  PROC DrawPart118()
    MoveL Offs(pOrigin,175.68,196.88,0.00),v40,fine,tPen\WObj:=wPaper;
    MoveL Offs(pOrigin,175.68,196.88,6.00),v60,z5,tPen\WObj:=wPaper;
    MoveL Offs(pOrigin,176.60,194.01,6.00),vTravel,z5,tPen\WObj:=wPaper;
    MoveL Offs(pOrigin,176.60,194.01,0.00),v60,z0,tPen\WObj:=wPaper;
    MoveL Offs(pOrigin,168.94,201.68,0.00),v40,z0,tPen\WObj:=wPaper;
    MoveL Offs(pOrigin,169.41,202.55,0.00),v40,z0,tPen\WObj:=wPaper;
    MoveL Offs(pOrigin,171.06,204.21,0.00),v40,fine,tPen\WObj:=wPaper;
    MoveL Offs(pOrigin,171.06,204.21,6.00),v60,z5,tPen\WObj:=wPaper;
    MoveL Offs(pOrigin,168.81,204.95,6.00),vTravel,z5,tPen\WObj:=wPaper;
    MoveL Offs(pOrigin,168.81,204.95,0.00),v60,z0,tPen\WObj:=wPaper;
    MoveL Offs(pOrigin,170.47,206.60,0.00),v40,z0,tPen\WObj:=wPaper;
    MoveL Offs(pOrigin,170.87,207.21,0.00),v40,z0,tPen\WObj:=wPaper;
    MoveL Offs(pOrigin,163.66,214.42,0.00),v40,z0,tPen\WObj:=wPaper;
    MoveL Offs(pOrigin,164.35,213.92,0.00),v40,z0,tPen\WObj:=wPaper;
    MoveL Offs(pOrigin,166.30,215.88,0.00),v40,fine,tPen\WObj:=wPaper;
    MoveL Offs(pOrigin,166.30,215.88,6.00),v60,z5,tPen\WObj:=wPaper;
    MoveL Offs(pOrigin,167.65,215.73,6.00),vTravel,z5,tPen\WObj:=wPaper;
    MoveL Offs(pOrigin,167.65,215.73,0.00),v60,z0,tPen\WObj:=wPaper;
    MoveL Offs(pOrigin,170.05,218.13,0.00),v40,z0,tPen\WObj:=wPaper;
    MoveL Offs(pOrigin,170.39,218.15,0.00),v40,z0,tPen\WObj:=wPaper;
    MoveL Offs(pOrigin,163.02,225.51,0.00),v40,z0,tPen\WObj:=wPaper;
    MoveL Offs(pOrigin,163.94,225.14,0.00),v40,z0,tPen\WObj:=wPaper;
    MoveL Offs(pOrigin,165.21,225.14,0.00),v40,z0,tPen\WObj:=wPaper;
    MoveL Offs(pOrigin,165.00,224.51,0.00),v40,z0,tPen\WObj:=wPaper;
    MoveL Offs(pOrigin,165.21,224.94,0.00),v40,z0,tPen\WObj:=wPaper;
    MoveL Offs(pOrigin,165.00,224.51,0.00),v40,z0,tPen\WObj:=wPaper;
    MoveL Offs(pOrigin,164.58,224.09,0.00),v40,z0,tPen\WObj:=wPaper;
    MoveL Offs(pOrigin,163.51,224.09,0.00),v40,z0,tPen\WObj:=wPaper;
    MoveL Offs(pOrigin,163.09,224.51,0.00),v40,z0,tPen\WObj:=wPaper;
    MoveL Offs(pOrigin,163.30,224.94,0.00),v40,z0,tPen\WObj:=wPaper;
    MoveL Offs(pOrigin,163.09,224.51,0.00),v40,z0,tPen\WObj:=wPaper;
    MoveL Offs(pOrigin,162.73,224.25,0.00),v40,z0,tPen\WObj:=wPaper;
    MoveL Offs(pOrigin,170.99,232.52,0.00),v40,z0,tPen\WObj:=wPaper;
    MoveL Offs(pOrigin,170.74,232.16,0.00),v40,z0,tPen\WObj:=wPaper;
    MoveL Offs(pOrigin,171.16,232.38,0.00),v40,z0,tPen\WObj:=wPaper;
    MoveL Offs(pOrigin,170.74,232.16,0.00),v40,z0,tPen\WObj:=wPaper;
    MoveL Offs(pOrigin,170.64,232.83,0.00),v40,z0,tPen\WObj:=wPaper;
    MoveL Offs(pOrigin,175.15,228.32,0.00),v40,z0,tPen\WObj:=wPaper;
    MoveL Offs(pOrigin,175.20,228.98,0.00),v40,z0,tPen\WObj:=wPaper;
    MoveL Offs(pOrigin,175.84,229.61,0.00),v40,z0,tPen\WObj:=wPaper;
    MoveL Offs(pOrigin,175.20,228.98,0.00),v40,z0,tPen\WObj:=wPaper;
    MoveL Offs(pOrigin,175.20,229.37,0.00),v40,z0,tPen\WObj:=wPaper;
    MoveL Offs(pOrigin,173.71,229.37,0.00),v40,z0,tPen\WObj:=wPaper;
    MoveL Offs(pOrigin,173.71,230.04,0.00),v40,z0,tPen\WObj:=wPaper;
    MoveL Offs(pOrigin,174.14,230.25,0.00),v40,z0,tPen\WObj:=wPaper;
    MoveL Offs(pOrigin,173.71,230.04,0.00),v40,z0,tPen\WObj:=wPaper;
    MoveL Offs(pOrigin,174.35,230.46,0.00),v40,z0,tPen\WObj:=wPaper;
    MoveL Offs(pOrigin,174.77,230.89,0.00),v40,z0,tPen\WObj:=wPaper;
    MoveL Offs(pOrigin,174.35,230.46,0.00),v40,z0,tPen\WObj:=wPaper;
    MoveL Offs(pOrigin,174.78,230.42,0.00),v40,z0,tPen\WObj:=wPaper;
    MoveL Offs(pOrigin,176.69,230.42,0.00),v40,z0,tPen\WObj:=wPaper;
    MoveL Offs(pOrigin,176.94,229.51,0.00),v40,z0,tPen\WObj:=wPaper;
    MoveL Offs(pOrigin,172.74,233.72,0.00),v40,z0,tPen\WObj:=wPaper;
    MoveL Offs(pOrigin,173.71,233.65,0.00),v40,z0,tPen\WObj:=wPaper;
    MoveL Offs(pOrigin,174.14,233.86,0.00),v40,z0,tPen\WObj:=wPaper;
    MoveL Offs(pOrigin,173.71,233.65,0.00),v40,z0,tPen\WObj:=wPaper;
    MoveL Offs(pOrigin,173.63,234.32,0.00),v40,z0,tPen\WObj:=wPaper;
    MoveL Offs(pOrigin,177.84,230.11,0.00),v40,z0,tPen\WObj:=wPaper;
    MoveL Offs(pOrigin,178.74,230.71,0.00),v40,z0,tPen\WObj:=wPaper;
    MoveL Offs(pOrigin,174.68,234.76,0.00),v40,z0,tPen\WObj:=wPaper;
    MoveL Offs(pOrigin,174.15,234.18,0.00),v40,z0,tPen\WObj:=wPaper;
    MoveL Offs(pOrigin,161.22,221.25,0.00),v40,z0,tPen\WObj:=wPaper;
    MoveL Offs(pOrigin,161.09,221.47,0.00),v40,z0,tPen\WObj:=wPaper;
    MoveL Offs(pOrigin,170.25,212.31,0.00),v40,z0,tPen\WObj:=wPaper;
    MoveL Offs(pOrigin,169.88,211.99,0.00),v40,z0,tPen\WObj:=wPaper;
    MoveL Offs(pOrigin,168.08,210.19,0.00),v40,fine,tPen\WObj:=wPaper;
    MoveL Offs(pOrigin,168.08,210.19,6.00),v60,z5,tPen\WObj:=wPaper;
    MoveL Offs(pOrigin,167.93,211.54,6.00),vTravel,z5,tPen\WObj:=wPaper;
    MoveL Offs(pOrigin,167.93,211.54,0.00),v60,z0,tPen\WObj:=wPaper;
    MoveL Offs(pOrigin,169.89,213.49,0.00),v40,z0,tPen\WObj:=wPaper;
    MoveL Offs(pOrigin,170.25,213.81,0.00),v40,z0,tPen\WObj:=wPaper;
    MoveL Offs(pOrigin,161.38,222.67,0.00),v40,fine,tPen\WObj:=wPaper;
    MoveL Offs(pOrigin,161.38,222.67,6.00),v60,z5,tPen\WObj:=wPaper;
    MoveL Offs(pOrigin,162.45,221.98,6.00),vTravel,z5,tPen\WObj:=wPaper;
    MoveL Offs(pOrigin,162.45,221.98,0.00),v60,z0,tPen\WObj:=wPaper;
    MoveL Offs(pOrigin,163.51,221.98,0.00),v40,z0,tPen\WObj:=wPaper;
    MoveL Offs(pOrigin,163.09,220.92,0.00),v40,z0,tPen\WObj:=wPaper;
    MoveL Offs(pOrigin,162.02,220.92,0.00),v40,fine,tPen\WObj:=wPaper;
    MoveL Offs(pOrigin,162.02,220.92,6.00),v60,z5,tPen\WObj:=wPaper;
    MoveL Offs(pOrigin,165.27,220.82,6.00),vTravel,z5,tPen\WObj:=wPaper;
    MoveL Offs(pOrigin,165.27,220.82,0.00),v60,z0,tPen\WObj:=wPaper;
    MoveL Offs(pOrigin,168.12,223.67,0.00),v40,fine,tPen\WObj:=wPaper;
    MoveL Offs(pOrigin,168.12,223.67,6.00),v60,z5,tPen\WObj:=wPaper;
    MoveL Offs(pOrigin,166.70,223.45,6.00),vTravel,z5,tPen\WObj:=wPaper;
    MoveL Offs(pOrigin,166.70,223.45,0.00),v60,z0,tPen\WObj:=wPaper;
    MoveL Offs(pOrigin,166.91,223.88,0.00),v40,z0,tPen\WObj:=wPaper;
    MoveL Offs(pOrigin,166.70,223.45,0.00),v40,z0,tPen\WObj:=wPaper;
    MoveL Offs(pOrigin,165.87,222.91,0.00),v40,z0,tPen\WObj:=wPaper;
    MoveL Offs(pOrigin,168.73,225.77,0.00),v40,z0,tPen\WObj:=wPaper;
    MoveL Offs(pOrigin,168.40,225.79,0.00),v40,z0,tPen\WObj:=wPaper;
    MoveL Offs(pOrigin,168.40,224.94,0.00),v40,z0,tPen\WObj:=wPaper;
    MoveL Offs(pOrigin,166.91,221.11,0.00),v40,z0,tPen\WObj:=wPaper;
    MoveL Offs(pOrigin,166.06,216.86,0.00),v40,z0,tPen\WObj:=wPaper;
    MoveL Offs(pOrigin,165.85,209.64,0.00),v40,z0,tPen\WObj:=wPaper;
    MoveL Offs(pOrigin,166.70,202.20,0.00),v40,z0,tPen\WObj:=wPaper;
    MoveL Offs(pOrigin,168.26,196.32,0.00),v40,z0,tPen\WObj:=wPaper;
    MoveL Offs(pOrigin,168.61,196.25,0.00),v40,z0,tPen\WObj:=wPaper;
    MoveL Offs(pOrigin,171.16,197.31,0.00),v40,z0,tPen\WObj:=wPaper;
    MoveL Offs(pOrigin,169.04,205.18,0.00),v40,z0,tPen\WObj:=wPaper;
    MoveL Offs(pOrigin,167.98,212.82,0.00),v40,z0,tPen\WObj:=wPaper;
    MoveL Offs(pOrigin,168.19,217.93,0.00),v40,z0,tPen\WObj:=wPaper;
    MoveL Offs(pOrigin,169.60,223.88,0.00),v40,z0,tPen\WObj:=wPaper;
    MoveL Offs(pOrigin,171.80,227.70,0.00),v40,z0,tPen\WObj:=wPaper;
    MoveL Offs(pOrigin,174.77,230.68,0.00),v40,z0,tPen\WObj:=wPaper;
    MoveL Offs(pOrigin,178.81,232.87,0.00),v40,z0,tPen\WObj:=wPaper;
    MoveL Offs(pOrigin,182.85,234.07,0.00),v40,z0,tPen\WObj:=wPaper;
    MoveL Offs(pOrigin,183.70,233.86,0.00),v40,z0,tPen\WObj:=wPaper;
    MoveL Offs(pOrigin,183.70,233.86,0.00),v40,z0,tPen\WObj:=wPaper;
    MoveL Offs(pOrigin,186.68,234.50,0.00),v40,z0,tPen\WObj:=wPaper;
    MoveL Offs(pOrigin,186.66,234.73,0.00),v40,z0,tPen\WObj:=wPaper;
    MoveL Offs(pOrigin,183.81,237.58,0.00),v40,z0,tPen\WObj:=wPaper;
    MoveL Offs(pOrigin,184.34,236.76,0.00),v40,z0,tPen\WObj:=wPaper;
    MoveL Offs(pOrigin,189.86,236.76,0.00),v40,z0,tPen\WObj:=wPaper;
    MoveL Offs(pOrigin,189.88,236.47,0.00),v40,z0,tPen\WObj:=wPaper;
    MoveL Offs(pOrigin,192.44,239.02,0.00),v40,z0,tPen\WObj:=wPaper;
    MoveL Offs(pOrigin,192.49,239.35,0.00),v40,z0,tPen\WObj:=wPaper;
    MoveL Offs(pOrigin,195.05,236.80,0.00),v40,z0,tPen\WObj:=wPaper;
    MoveL Offs(pOrigin,195.43,237.54,0.00),v40,z0,tPen\WObj:=wPaper;
    MoveL Offs(pOrigin,197.98,240.09,0.00),v40,z0,tPen\WObj:=wPaper;
    MoveL Offs(pOrigin,197.43,240.39,0.00),v40,z0,tPen\WObj:=wPaper;
  ENDPROC

  PROC DrawPart119()
    MoveL Offs(pOrigin,204.49,233.32,0.00),v40,z0,tPen\WObj:=wPaper;
    MoveL Offs(pOrigin,204.10,232.77,0.00),v40,z0,tPen\WObj:=wPaper;
    MoveL Offs(pOrigin,202.30,230.97,0.00),v40,z0,tPen\WObj:=wPaper;
    MoveL Offs(pOrigin,203.04,230.42,0.00),v40,z0,tPen\WObj:=wPaper;
    MoveL Offs(pOrigin,204.10,230.42,0.00),v40,z0,tPen\WObj:=wPaper;
    MoveL Offs(pOrigin,204.69,230.37,0.00),v40,z0,tPen\WObj:=wPaper;
    MoveL Offs(pOrigin,203.34,229.02,0.00),v40,z0,tPen\WObj:=wPaper;
    MoveL Offs(pOrigin,203.46,229.37,0.00),v40,z0,tPen\WObj:=wPaper;
    MoveL Offs(pOrigin,204.74,229.37,0.00),v40,z0,tPen\WObj:=wPaper;
    MoveL Offs(pOrigin,205.38,228.76,0.00),v40,z0,tPen\WObj:=wPaper;
    MoveL Offs(pOrigin,204.74,229.40,0.00),v40,z0,tPen\WObj:=wPaper;
    MoveL Offs(pOrigin,205.38,228.76,0.00),v40,fine,tPen\WObj:=wPaper;
    MoveL Offs(pOrigin,205.38,228.76,6.00),v60,z5,tPen\WObj:=wPaper;
    MoveL Offs(pOrigin,204.31,227.91,6.00),vTravel,z5,tPen\WObj:=wPaper;
    MoveL Offs(pOrigin,204.31,227.91,0.00),v60,z0,tPen\WObj:=wPaper;
    MoveL Offs(pOrigin,203.89,228.34,0.00),v40,z0,tPen\WObj:=wPaper;
    MoveL Offs(pOrigin,204.31,227.91,0.00),v40,z0,tPen\WObj:=wPaper;
    MoveL Offs(pOrigin,204.68,227.38,0.00),v40,z0,tPen\WObj:=wPaper;
    MoveL Offs(pOrigin,208.44,231.13,0.00),v40,z0,tPen\WObj:=wPaper;
    MoveL Offs(pOrigin,208.69,232.11,0.00),v40,z0,tPen\WObj:=wPaper;
    MoveL Offs(pOrigin,205.99,234.82,0.00),v40,fine,tPen\WObj:=wPaper;
    MoveL Offs(pOrigin,205.99,234.82,6.00),v60,z5,tPen\WObj:=wPaper;
    MoveL Offs(pOrigin,205.98,236.32,6.00),vTravel,z5,tPen\WObj:=wPaper;
    MoveL Offs(pOrigin,205.98,236.32,0.00),v60,z0,tPen\WObj:=wPaper;
    MoveL Offs(pOrigin,208.24,234.06,0.00),v40,z0,tPen\WObj:=wPaper;
    MoveL Offs(pOrigin,207.85,233.53,0.00),v40,z0,tPen\WObj:=wPaper;
    MoveL Offs(pOrigin,206.95,232.63,0.00),v40,z0,tPen\WObj:=wPaper;
    MoveL Offs(pOrigin,207.29,232.38,0.00),v40,z0,tPen\WObj:=wPaper;
    MoveL Offs(pOrigin,207.71,228.76,0.00),v40,z0,tPen\WObj:=wPaper;
    MoveL Offs(pOrigin,207.29,228.34,0.00),v40,z0,tPen\WObj:=wPaper;
    MoveL Offs(pOrigin,206.44,228.34,0.00),v40,z0,tPen\WObj:=wPaper;
    MoveL Offs(pOrigin,204.95,229.40,0.00),v40,z0,tPen\WObj:=wPaper;
    MoveL Offs(pOrigin,204.03,231.10,0.00),v40,z0,tPen\WObj:=wPaper;
    MoveL Offs(pOrigin,203.68,232.38,0.00),v40,z0,tPen\WObj:=wPaper;
    MoveL Offs(pOrigin,203.46,236.41,0.00),v40,z0,tPen\WObj:=wPaper;
    MoveL Offs(pOrigin,202.47,240.66,0.00),v40,z0,tPen\WObj:=wPaper;
    MoveL Offs(pOrigin,200.98,244.91,0.00),v40,z0,tPen\WObj:=wPaper;
    MoveL Offs(pOrigin,196.80,252.14,0.00),v40,z0,tPen\WObj:=wPaper;
    MoveL Offs(pOrigin,196.24,254.48,0.00),v40,z0,tPen\WObj:=wPaper;
    MoveL Offs(pOrigin,196.24,258.30,0.00),v40,z0,tPen\WObj:=wPaper;
    MoveL Offs(pOrigin,196.80,260.42,0.00),v40,z0,tPen\WObj:=wPaper;
    MoveL Offs(pOrigin,197.73,262.12,0.00),v40,z0,tPen\WObj:=wPaper;
    MoveL Offs(pOrigin,199.00,263.12,0.00),v40,z0,tPen\WObj:=wPaper;
    MoveL Offs(pOrigin,200.70,263.19,0.00),v40,z0,tPen\WObj:=wPaper;
    MoveL Offs(pOrigin,201.98,261.91,0.00),v40,z0,tPen\WObj:=wPaper;
    MoveL Offs(pOrigin,201.98,261.91,0.00),v40,z0,tPen\WObj:=wPaper;
    MoveL Offs(pOrigin,202.54,261.70,0.00),v40,z0,tPen\WObj:=wPaper;
    MoveL Offs(pOrigin,202.90,260.00,0.00),v40,z0,tPen\WObj:=wPaper;
    MoveL Offs(pOrigin,203.46,259.36,0.00),v40,z0,tPen\WObj:=wPaper;
    MoveL Offs(pOrigin,203.68,258.09,0.00),v40,z0,tPen\WObj:=wPaper;
    MoveL Offs(pOrigin,203.39,257.02,0.00),v40,z0,tPen\WObj:=wPaper;
    MoveL Offs(pOrigin,204.38,252.14,0.00),v40,z0,tPen\WObj:=wPaper;
    MoveL Offs(pOrigin,205.02,250.44,0.00),v40,z0,tPen\WObj:=wPaper;
    MoveL Offs(pOrigin,205.80,250.65,0.00),v40,z0,tPen\WObj:=wPaper;
    MoveL Offs(pOrigin,205.93,250.44,0.00),v40,z0,tPen\WObj:=wPaper;
    MoveL Offs(pOrigin,205.93,260.42,0.00),v40,z0,tPen\WObj:=wPaper;
    MoveL Offs(pOrigin,206.23,260.85,0.00),v40,z0,tPen\WObj:=wPaper;
    MoveL Offs(pOrigin,206.01,261.27,0.00),v40,z0,tPen\WObj:=wPaper;
    MoveL Offs(pOrigin,206.23,260.85,0.00),v40,z0,tPen\WObj:=wPaper;
    MoveL Offs(pOrigin,206.01,261.05,0.00),v40,z0,tPen\WObj:=wPaper;
    MoveL Offs(pOrigin,203.04,261.05,0.00),v40,z0,tPen\WObj:=wPaper;
    MoveL Offs(pOrigin,203.04,259.99,0.00),v40,z0,tPen\WObj:=wPaper;
    MoveL Offs(pOrigin,207.29,259.99,0.00),v40,z0,tPen\WObj:=wPaper;
    MoveL Offs(pOrigin,207.78,260.34,0.00),v40,z0,tPen\WObj:=wPaper;
    MoveL Offs(pOrigin,203.12,255.69,0.00),v40,z0,tPen\WObj:=wPaper;
    MoveL Offs(pOrigin,203.68,255.77,0.00),v40,z0,tPen\WObj:=wPaper;
    MoveL Offs(pOrigin,207.08,255.77,0.00),v40,z0,tPen\WObj:=wPaper;
    MoveL Offs(pOrigin,207.08,254.71,0.00),v40,z0,tPen\WObj:=wPaper;
    MoveL Offs(pOrigin,203.89,254.71,0.00),v40,z0,tPen\WObj:=wPaper;
    MoveL Offs(pOrigin,203.42,254.49,0.00),v40,z0,tPen\WObj:=wPaper;
    MoveL Offs(pOrigin,208.23,259.30,0.00),v40,z0,tPen\WObj:=wPaper;
    MoveL Offs(pOrigin,207.93,258.94,0.00),v40,z0,tPen\WObj:=wPaper;
    MoveL Offs(pOrigin,207.07,258.73,0.00),v40,z0,tPen\WObj:=wPaper;
    MoveL Offs(pOrigin,207.29,257.88,0.00),v40,z0,tPen\WObj:=wPaper;
    MoveL Offs(pOrigin,207.07,257.88,0.00),v40,z0,tPen\WObj:=wPaper;
    MoveL Offs(pOrigin,207.50,257.88,0.00),v40,z0,tPen\WObj:=wPaper;
    MoveL Offs(pOrigin,203.04,257.88,0.00),v40,z0,tPen\WObj:=wPaper;
    MoveL Offs(pOrigin,203.25,257.45,0.00),v40,z0,tPen\WObj:=wPaper;
    MoveL Offs(pOrigin,202.12,258.51,0.00),v40,z0,tPen\WObj:=wPaper;
    MoveL Offs(pOrigin,201.98,259.79,0.00),v40,z0,tPen\WObj:=wPaper;
    MoveL Offs(pOrigin,202.61,258.94,0.00),v40,z0,tPen\WObj:=wPaper;
    MoveL Offs(pOrigin,207.50,258.94,0.00),v40,fine,tPen\WObj:=wPaper;
    MoveL Offs(pOrigin,207.50,258.94,6.00),v60,z5,tPen\WObj:=wPaper;
    MoveL Offs(pOrigin,208.76,258.93,6.00),vTravel,z5,tPen\WObj:=wPaper;
    MoveL Offs(pOrigin,208.76,258.93,0.00),v60,z0,tPen\WObj:=wPaper;
    MoveL Offs(pOrigin,194.18,273.50,0.00),v40,z0,tPen\WObj:=wPaper;
    MoveL Offs(pOrigin,194.64,274.08,0.00),v40,z0,tPen\WObj:=wPaper;
    MoveL Offs(pOrigin,204.71,284.15,0.00),v40,z0,tPen\WObj:=wPaper;
    MoveL Offs(pOrigin,204.31,284.28,0.00),v40,z0,tPen\WObj:=wPaper;
    MoveL Offs(pOrigin,191.35,284.28,0.00),v40,z0,tPen\WObj:=wPaper;
    MoveL Offs(pOrigin,190.93,283.81,0.00),v40,z0,tPen\WObj:=wPaper;
    MoveL Offs(pOrigin,195.58,288.47,0.00),v40,fine,tPen\WObj:=wPaper;
    MoveL Offs(pOrigin,195.58,288.47,6.00),v60,z5,tPen\WObj:=wPaper;
    MoveL Offs(pOrigin,193.90,289.54,6.00),vTravel,z5,tPen\WObj:=wPaper;
    MoveL Offs(pOrigin,193.90,289.54,0.00),v60,z0,tPen\WObj:=wPaper;
    MoveL Offs(pOrigin,194.11,289.96,0.00),v40,z0,tPen\WObj:=wPaper;
    MoveL Offs(pOrigin,193.90,289.54,0.00),v40,z0,tPen\WObj:=wPaper;
    MoveL Offs(pOrigin,193.48,289.56,0.00),v40,z0,tPen\WObj:=wPaper;
    MoveL Offs(pOrigin,191.56,289.56,0.00),v40,z0,tPen\WObj:=wPaper;
    MoveL Offs(pOrigin,191.09,289.95,0.00),v40,z0,tPen\WObj:=wPaper;
    MoveL Offs(pOrigin,196.20,295.06,0.00),v40,z0,tPen\WObj:=wPaper;
    MoveL Offs(pOrigin,196.45,295.49,0.00),v40,z0,tPen\WObj:=wPaper;
    MoveL Offs(pOrigin,197.51,297.19,0.00),v40,z0,tPen\WObj:=wPaper;
    MoveL Offs(pOrigin,199.64,299.31,0.00),v40,z0,tPen\WObj:=wPaper;
    MoveL Offs(pOrigin,200.71,299.57,0.00),v40,z0,tPen\WObj:=wPaper;
    MoveL Offs(pOrigin,225.80,324.66,0.00),v40,fine,tPen\WObj:=wPaper;
    MoveL Offs(pOrigin,225.80,324.66,6.00),v60,z5,tPen\WObj:=wPaper;
    MoveL Offs(pOrigin,225.95,323.31,6.00),vTravel,z5,tPen\WObj:=wPaper;
    MoveL Offs(pOrigin,225.95,323.31,0.00),v60,z0,tPen\WObj:=wPaper;
    MoveL Offs(pOrigin,201.76,299.12,0.00),v40,z0,tPen\WObj:=wPaper;
    MoveL Offs(pOrigin,202.40,299.95,0.00),v40,z0,tPen\WObj:=wPaper;
    MoveL Offs(pOrigin,204.95,301.01,0.00),v40,z0,tPen\WObj:=wPaper;
    MoveL Offs(pOrigin,204.88,300.80,0.00),v40,z0,tPen\WObj:=wPaper;
    MoveL Offs(pOrigin,204.88,301.86,0.00),v40,fine,tPen\WObj:=wPaper;
    MoveL Offs(pOrigin,204.88,301.86,6.00),v60,z5,tPen\WObj:=wPaper;
    MoveL Offs(pOrigin,203.68,302.23,6.00),vTravel,z5,tPen\WObj:=wPaper;
    MoveL Offs(pOrigin,203.68,302.23,0.00),v60,z0,tPen\WObj:=wPaper;
    MoveL Offs(pOrigin,210.48,302.23,0.00),v40,fine,tPen\WObj:=wPaper;
    MoveL Offs(pOrigin,210.48,302.23,6.00),v60,z5,tPen\WObj:=wPaper;
    MoveL Offs(pOrigin,211.33,301.16,6.00),vTravel,z5,tPen\WObj:=wPaper;
  ENDPROC

  PROC DrawPart120()
    MoveL Offs(pOrigin,211.33,301.16,0.00),v60,z0,tPen\WObj:=wPaper;
    MoveL Offs(pOrigin,195.70,316.79,0.00),v40,z0,tPen\WObj:=wPaper;
    MoveL Offs(pOrigin,196.45,317.59,0.00),v40,z0,tPen\WObj:=wPaper;
    MoveL Offs(pOrigin,196.66,318.01,0.00),v40,z0,tPen\WObj:=wPaper;
    MoveL Offs(pOrigin,196.45,317.59,0.00),v40,z0,tPen\WObj:=wPaper;
    MoveL Offs(pOrigin,196.15,317.84,0.00),v40,z0,tPen\WObj:=wPaper;
    MoveL Offs(pOrigin,212.07,301.91,0.00),v40,z0,tPen\WObj:=wPaper;
    MoveL Offs(pOrigin,212.82,302.66,0.00),v40,z0,tPen\WObj:=wPaper;
    MoveL Offs(pOrigin,202.60,312.87,0.00),v40,z0,tPen\WObj:=wPaper;
    MoveL Offs(pOrigin,203.05,313.92,0.00),v40,z0,tPen\WObj:=wPaper;
    MoveL Offs(pOrigin,197.34,319.63,0.00),v40,z0,tPen\WObj:=wPaper;
    MoveL Offs(pOrigin,197.73,319.50,0.00),v40,z0,tPen\WObj:=wPaper;
    MoveL Offs(pOrigin,198.15,319.92,0.00),v40,z0,tPen\WObj:=wPaper;
    MoveL Offs(pOrigin,197.73,319.50,0.00),v40,z0,tPen\WObj:=wPaper;
    MoveL Offs(pOrigin,198.15,319.13,0.00),v40,z0,tPen\WObj:=wPaper;
    MoveL Offs(pOrigin,199.42,319.13,0.00),v40,z0,tPen\WObj:=wPaper;
    MoveL Offs(pOrigin,199.43,319.08,0.00),v40,z0,tPen\WObj:=wPaper;
    MoveL Offs(pOrigin,200.06,319.71,0.00),v40,z0,tPen\WObj:=wPaper;
    MoveL Offs(pOrigin,199.43,319.08,0.00),v40,z0,tPen\WObj:=wPaper;
    MoveL Offs(pOrigin,199.00,320.18,0.00),v40,z0,tPen\WObj:=wPaper;
    MoveL Offs(pOrigin,200.91,320.18,0.00),v40,z0,tPen\WObj:=wPaper;
    MoveL Offs(pOrigin,200.70,320.14,0.00),v40,z0,tPen\WObj:=wPaper;
    MoveL Offs(pOrigin,201.12,320.35,0.00),v40,z0,tPen\WObj:=wPaper;
    MoveL Offs(pOrigin,200.70,320.14,0.00),v40,fine,tPen\WObj:=wPaper;
    MoveL Offs(pOrigin,200.70,320.14,6.00),v60,z5,tPen\WObj:=wPaper;
    MoveL Offs(pOrigin,199.85,321.24,6.00),vTravel,z5,tPen\WObj:=wPaper;
    MoveL Offs(pOrigin,199.85,321.24,0.00),v60,z0,tPen\WObj:=wPaper;
    MoveL Offs(pOrigin,202.40,321.24,0.00),v40,z0,tPen\WObj:=wPaper;
    MoveL Offs(pOrigin,202.61,321.41,0.00),v40,z0,tPen\WObj:=wPaper;
    MoveL Offs(pOrigin,204.10,321.13,0.00),v40,z0,tPen\WObj:=wPaper;
    MoveL Offs(pOrigin,205.38,321.62,0.00),v40,z0,tPen\WObj:=wPaper;
    MoveL Offs(pOrigin,205.45,321.41,0.00),v40,z0,tPen\WObj:=wPaper;
    MoveL Offs(pOrigin,206.65,320.56,0.00),v40,z0,tPen\WObj:=wPaper;
    MoveL Offs(pOrigin,209.34,320.35,0.00),v40,z0,tPen\WObj:=wPaper;
    MoveL Offs(pOrigin,208.56,321.41,0.00),v40,z0,tPen\WObj:=wPaper;
    MoveL Offs(pOrigin,206.23,321.84,0.00),v40,z0,tPen\WObj:=wPaper;
    MoveL Offs(pOrigin,205.45,321.41,0.00),v40,z0,tPen\WObj:=wPaper;
    MoveL Offs(pOrigin,205.38,320.99,0.00),v40,z0,tPen\WObj:=wPaper;
    MoveL Offs(pOrigin,204.10,320.85,0.00),v40,z0,tPen\WObj:=wPaper;
    MoveL Offs(pOrigin,203.46,320.21,0.00),v40,z0,tPen\WObj:=wPaper;
    MoveL Offs(pOrigin,200.63,318.65,0.00),v40,z0,tPen\WObj:=wPaper;
    MoveL Offs(pOrigin,200.49,317.80,0.00),v40,z0,tPen\WObj:=wPaper;
    MoveL Offs(pOrigin,200.49,317.80,0.00),v40,z0,tPen\WObj:=wPaper;
    MoveL Offs(pOrigin,201.76,318.01,0.00),v40,z0,tPen\WObj:=wPaper;
    MoveL Offs(pOrigin,201.76,318.01,0.00),v40,z0,tPen\WObj:=wPaper;
    MoveL Offs(pOrigin,202.40,319.08,0.00),v40,z0,tPen\WObj:=wPaper;
    MoveL Offs(pOrigin,202.40,319.50,0.00),v40,z0,tPen\WObj:=wPaper;
    MoveL Offs(pOrigin,203.04,319.08,0.00),v40,z0,tPen\WObj:=wPaper;
    MoveL Offs(pOrigin,206.01,320.00,0.00),v40,z0,tPen\WObj:=wPaper;
    MoveL Offs(pOrigin,206.44,320.56,0.00),v40,z0,tPen\WObj:=wPaper;
    MoveL Offs(pOrigin,206.33,319.60,0.00),v40,z0,tPen\WObj:=wPaper;
    MoveL Offs(pOrigin,201.67,324.26,0.00),v40,z0,tPen\WObj:=wPaper;
    MoveL Offs(pOrigin,200.92,323.51,0.00),v40,z0,tPen\WObj:=wPaper;
    MoveL Offs(pOrigin,217.60,306.84,0.00),v40,z0,tPen\WObj:=wPaper;
    MoveL Offs(pOrigin,217.66,307.56,0.00),v40,z0,tPen\WObj:=wPaper;
    MoveL Offs(pOrigin,234.19,324.09,0.00),v40,z0,tPen\WObj:=wPaper;
    MoveL Offs(pOrigin,234.70,323.35,0.00),v40,z0,tPen\WObj:=wPaper;
    MoveL Offs(pOrigin,239.16,323.35,0.00),v40,z0,tPen\WObj:=wPaper;
    MoveL Offs(pOrigin,239.59,323.11,0.00),v40,z0,tPen\WObj:=wPaper;
    MoveL Offs(pOrigin,237.04,320.77,0.00),v40,z0,tPen\WObj:=wPaper;
    MoveL Offs(pOrigin,237.04,320.77,0.00),v40,z0,tPen\WObj:=wPaper;
    MoveL Offs(pOrigin,235.76,321.41,0.00),v40,z0,tPen\WObj:=wPaper;
    MoveL Offs(pOrigin,235.55,322.05,0.00),v40,z0,tPen\WObj:=wPaper;
    MoveL Offs(pOrigin,235.55,322.05,0.00),v40,z0,tPen\WObj:=wPaper;
    MoveL Offs(pOrigin,237.89,325.66,0.00),v40,z0,tPen\WObj:=wPaper;
    MoveL Offs(pOrigin,238.52,325.46,0.00),v40,z0,tPen\WObj:=wPaper;
    MoveL Offs(pOrigin,240.22,325.46,0.00),v40,z0,tPen\WObj:=wPaper;
    MoveL Offs(pOrigin,239.59,325.88,0.00),v40,z0,tPen\WObj:=wPaper;
    MoveL Offs(pOrigin,241.22,326.94,0.00),v40,z0,tPen\WObj:=wPaper;
    MoveL Offs(pOrigin,241.50,328.00,0.00),v40,z0,tPen\WObj:=wPaper;
    MoveL Offs(pOrigin,241.50,329.70,0.00),v40,z0,tPen\WObj:=wPaper;
    MoveL Offs(pOrigin,240.65,330.76,0.00),v40,z0,tPen\WObj:=wPaper;
    MoveL Offs(pOrigin,240.65,330.76,0.00),v40,z0,tPen\WObj:=wPaper;
    MoveL Offs(pOrigin,240.58,331.75,0.00),v40,z0,tPen\WObj:=wPaper;
    MoveL Offs(pOrigin,238.31,333.31,0.00),v40,z0,tPen\WObj:=wPaper;
    MoveL Offs(pOrigin,238.31,333.31,0.00),v40,z0,tPen\WObj:=wPaper;
    MoveL Offs(pOrigin,237.96,334.80,0.00),v40,z0,tPen\WObj:=wPaper;
    MoveL Offs(pOrigin,237.04,335.37,0.00),v40,z0,tPen\WObj:=wPaper;
    MoveL Offs(pOrigin,234.06,336.29,0.00),v40,z0,tPen\WObj:=wPaper;
    MoveL Offs(pOrigin,229.39,336.71,0.00),v40,z0,tPen\WObj:=wPaper;
    MoveL Offs(pOrigin,227.19,337.35,0.00),v40,z0,tPen\WObj:=wPaper;
    MoveL Offs(pOrigin,227.48,337.99,0.00),v40,z0,tPen\WObj:=wPaper;
    MoveL Offs(pOrigin,228.32,338.41,0.00),v40,z0,tPen\WObj:=wPaper;
    MoveL Offs(pOrigin,231.30,338.41,0.00),v40,z0,tPen\WObj:=wPaper;
    MoveL Offs(pOrigin,232.15,338.84,0.00),v40,z0,tPen\WObj:=wPaper;
    MoveL Offs(pOrigin,235.12,338.84,0.00),v40,z0,tPen\WObj:=wPaper;
    MoveL Offs(pOrigin,236.40,338.41,0.00),v40,z0,tPen\WObj:=wPaper;
    MoveL Offs(pOrigin,236.40,338.41,0.00),v40,z0,tPen\WObj:=wPaper;
    MoveL Offs(pOrigin,237.25,338.62,0.00),v40,z0,tPen\WObj:=wPaper;
    MoveL Offs(pOrigin,240.01,337.99,0.00),v40,z0,tPen\WObj:=wPaper;
    MoveL Offs(pOrigin,242.77,336.85,0.00),v40,z0,tPen\WObj:=wPaper;
    MoveL Offs(pOrigin,243.84,335.79,0.00),v40,z0,tPen\WObj:=wPaper;
    MoveL Offs(pOrigin,244.90,336.00,0.00),v40,z0,tPen\WObj:=wPaper;
    MoveL Offs(pOrigin,245.82,335.51,0.00),v40,z0,tPen\WObj:=wPaper;
    MoveL Offs(pOrigin,245.54,335.65,0.00),v40,z0,tPen\WObj:=wPaper;
    MoveL Offs(pOrigin,245.75,336.02,0.00),v40,z0,tPen\WObj:=wPaper;
    MoveL Offs(pOrigin,247.02,336.02,0.00),v40,z0,tPen\WObj:=wPaper;
    MoveL Offs(pOrigin,247.24,336.50,0.00),v40,z0,tPen\WObj:=wPaper;
    MoveL Offs(pOrigin,248.65,335.65,0.00),v40,z0,tPen\WObj:=wPaper;
    MoveL Offs(pOrigin,249.15,334.59,0.00),v40,z0,tPen\WObj:=wPaper;
    MoveL Offs(pOrigin,249.50,334.92,0.00),v40,z0,tPen\WObj:=wPaper;
    MoveL Offs(pOrigin,248.30,333.72,0.00),v40,z0,tPen\WObj:=wPaper;
    MoveL Offs(pOrigin,249.15,333.95,0.00),v40,z0,tPen\WObj:=wPaper;
    MoveL Offs(pOrigin,248.94,332.89,0.00),v40,z0,tPen\WObj:=wPaper;
    MoveL Offs(pOrigin,250.00,329.70,0.00),v40,z0,tPen\WObj:=wPaper;
    MoveL Offs(pOrigin,249.57,328.85,0.00),v40,z0,tPen\WObj:=wPaper;
    MoveL Offs(pOrigin,249.22,326.30,0.00),v40,z0,tPen\WObj:=wPaper;
    MoveL Offs(pOrigin,248.16,325.02,0.00),v40,z0,tPen\WObj:=wPaper;
    MoveL Offs(pOrigin,248.09,324.17,0.00),v40,z0,tPen\WObj:=wPaper;
    MoveL Offs(pOrigin,248.09,324.17,0.00),v40,z0,tPen\WObj:=wPaper;
    MoveL Offs(pOrigin,248.09,323.75,0.00),v40,z0,tPen\WObj:=wPaper;
    MoveL Offs(pOrigin,248.51,323.54,0.00),v40,z0,tPen\WObj:=wPaper;
    MoveL Offs(pOrigin,248.09,324.17,0.00),v40,z0,tPen\WObj:=wPaper;
    MoveL Offs(pOrigin,246.39,323.75,0.00),v40,z0,tPen\WObj:=wPaper;
    MoveL Offs(pOrigin,246.39,323.96,0.00),v40,z0,tPen\WObj:=wPaper;
    MoveL Offs(pOrigin,246.39,323.96,0.00),v40,z0,tPen\WObj:=wPaper;
    MoveL Offs(pOrigin,245.11,322.55,0.00),v40,z0,tPen\WObj:=wPaper;
    MoveL Offs(pOrigin,243.41,322.12,0.00),v40,z0,tPen\WObj:=wPaper;
    MoveL Offs(pOrigin,243.20,322.48,0.00),v40,z0,tPen\WObj:=wPaper;
    MoveL Offs(pOrigin,243.70,323.96,0.00),v40,z0,tPen\WObj:=wPaper;
  ENDPROC

  PROC DrawPart121()
    MoveL Offs(pOrigin,244.69,325.24,0.00),v40,z0,tPen\WObj:=wPaper;
    MoveL Offs(pOrigin,244.69,325.24,0.00),v40,z0,tPen\WObj:=wPaper;
    MoveL Offs(pOrigin,245.32,328.00,0.00),v40,z0,tPen\WObj:=wPaper;
    MoveL Offs(pOrigin,245.11,332.89,0.00),v40,z0,tPen\WObj:=wPaper;
    MoveL Offs(pOrigin,245.11,332.89,0.00),v40,z0,tPen\WObj:=wPaper;
    MoveL Offs(pOrigin,246.25,331.83,0.00),v40,z0,tPen\WObj:=wPaper;
    MoveL Offs(pOrigin,246.81,329.91,0.00),v40,z0,tPen\WObj:=wPaper;
    MoveL Offs(pOrigin,246.81,328.64,0.00),v40,z0,tPen\WObj:=wPaper;
    MoveL Offs(pOrigin,246.03,326.51,0.00),v40,z0,tPen\WObj:=wPaper;
    MoveL Offs(pOrigin,245.32,325.52,0.00),v40,z0,tPen\WObj:=wPaper;
    MoveL Offs(pOrigin,244.69,325.24,0.00),v40,z0,tPen\WObj:=wPaper;
    MoveL Offs(pOrigin,244.48,325.46,0.00),v40,z0,tPen\WObj:=wPaper;
    MoveL Offs(pOrigin,243.20,325.46,0.00),v40,z0,tPen\WObj:=wPaper;
    MoveL Offs(pOrigin,242.89,324.60,0.00),v40,z0,tPen\WObj:=wPaper;
    MoveL Offs(pOrigin,242.89,323.11,0.00),v40,z0,tPen\WObj:=wPaper;
    MoveL Offs(pOrigin,243.95,323.11,0.00),v40,z0,tPen\WObj:=wPaper;
    MoveL Offs(pOrigin,243.95,324.18,0.00),v40,fine,tPen\WObj:=wPaper;
    MoveL Offs(pOrigin,243.95,324.18,6.00),v60,z5,tPen\WObj:=wPaper;
    MoveL Offs(pOrigin,242.35,324.41,6.00),vTravel,z5,tPen\WObj:=wPaper;
    MoveL Offs(pOrigin,242.35,324.41,0.00),v60,z0,tPen\WObj:=wPaper;
    MoveL Offs(pOrigin,245.96,324.41,0.00),v40,z0,tPen\WObj:=wPaper;
    MoveL Offs(pOrigin,246.39,323.96,0.00),v40,z0,tPen\WObj:=wPaper;
    MoveL Offs(pOrigin,247.66,327.58,0.00),v40,z0,tPen\WObj:=wPaper;
    MoveL Offs(pOrigin,247.66,330.55,0.00),v40,z0,tPen\WObj:=wPaper;
    MoveL Offs(pOrigin,246.67,333.10,0.00),v40,z0,tPen\WObj:=wPaper;
    MoveL Offs(pOrigin,245.96,333.52,0.00),v40,z0,tPen\WObj:=wPaper;
    MoveL Offs(pOrigin,245.11,333.52,0.00),v40,z0,tPen\WObj:=wPaper;
    MoveL Offs(pOrigin,245.11,333.52,0.00),v40,z0,tPen\WObj:=wPaper;
    MoveL Offs(pOrigin,244.05,335.01,0.00),v40,z0,tPen\WObj:=wPaper;
    MoveL Offs(pOrigin,244.05,335.65,0.00),v40,z0,tPen\WObj:=wPaper;
    MoveL Offs(pOrigin,243.62,334.97,0.00),v40,z0,tPen\WObj:=wPaper;
    MoveL Offs(pOrigin,242.56,334.97,0.00),v40,z0,tPen\WObj:=wPaper;
    MoveL Offs(pOrigin,242.01,334.90,0.00),v40,z0,tPen\WObj:=wPaper;
    MoveL Offs(pOrigin,246.67,339.56,0.00),v40,z0,tPen\WObj:=wPaper;
    MoveL Offs(pOrigin,247.31,339.85,0.00),v40,z0,tPen\WObj:=wPaper;
    MoveL Offs(pOrigin,250.62,336.54,0.00),v40,z0,tPen\WObj:=wPaper;
    MoveL Offs(pOrigin,250.41,337.32,0.00),v40,z0,tPen\WObj:=wPaper;
    MoveL Offs(pOrigin,252.66,339.58,0.00),v40,z0,tPen\WObj:=wPaper;
    MoveL Offs(pOrigin,252.40,338.84,0.00),v40,z0,tPen\WObj:=wPaper;
    MoveL Offs(pOrigin,252.40,337.78,0.00),v40,z0,tPen\WObj:=wPaper;
    MoveL Offs(pOrigin,252.55,337.14,0.00),v40,z0,tPen\WObj:=wPaper;
    MoveL Offs(pOrigin,250.21,337.77,0.00),v40,z0,tPen\WObj:=wPaper;
    MoveL Offs(pOrigin,247.45,337.99,0.00),v40,z0,tPen\WObj:=wPaper;
    MoveL Offs(pOrigin,247.45,337.99,0.00),v40,z0,tPen\WObj:=wPaper;
    MoveL Offs(pOrigin,247.02,338.62,0.00),v40,z0,tPen\WObj:=wPaper;
    MoveL Offs(pOrigin,246.39,338.41,0.00),v40,z0,tPen\WObj:=wPaper;
    MoveL Offs(pOrigin,246.39,337.99,0.00),v40,z0,tPen\WObj:=wPaper;
    MoveL Offs(pOrigin,246.39,337.99,0.00),v40,z0,tPen\WObj:=wPaper;
    MoveL Offs(pOrigin,247.45,337.77,0.00),v40,z0,tPen\WObj:=wPaper;
    MoveL Offs(pOrigin,247.45,337.99,0.00),v40,z0,tPen\WObj:=wPaper;
    MoveL Offs(pOrigin,248.02,337.91,0.00),v40,z0,tPen\WObj:=wPaper;
    MoveL Offs(pOrigin,249.67,339.57,0.00),v40,z0,tPen\WObj:=wPaper;
    MoveL Offs(pOrigin,250.31,339.84,0.00),v40,z0,tPen\WObj:=wPaper;
    MoveL Offs(pOrigin,261.12,329.02,0.00),v40,z0,tPen\WObj:=wPaper;
    MoveL Offs(pOrigin,260.57,329.56,0.00),v40,z0,tPen\WObj:=wPaper;
    MoveL Offs(pOrigin,246.45,315.44,0.00),v40,z0,tPen\WObj:=wPaper;
    MoveL Offs(pOrigin,245.54,315.96,0.00),v40,z0,tPen\WObj:=wPaper;
    MoveL Offs(pOrigin,244.48,315.96,0.00),v40,z0,tPen\WObj:=wPaper;
    MoveL Offs(pOrigin,243.75,315.73,0.00),v40,z0,tPen\WObj:=wPaper;
    MoveL Offs(pOrigin,253.37,325.35,0.00),v40,z0,tPen\WObj:=wPaper;
    MoveL Offs(pOrigin,253.19,324.60,0.00),v40,z0,tPen\WObj:=wPaper;
    MoveL Offs(pOrigin,253.40,325.02,0.00),v40,z0,tPen\WObj:=wPaper;
    MoveL Offs(pOrigin,253.19,324.60,0.00),v40,fine,tPen\WObj:=wPaper;
    MoveL Offs(pOrigin,253.19,324.60,6.00),v60,z5,tPen\WObj:=wPaper;
    MoveL Offs(pOrigin,254.46,324.60,6.00),vTravel,z5,tPen\WObj:=wPaper;
    MoveL Offs(pOrigin,254.46,324.60,0.00),v60,z0,tPen\WObj:=wPaper;
    MoveL Offs(pOrigin,254.68,325.02,0.00),v40,z0,tPen\WObj:=wPaper;
    MoveL Offs(pOrigin,254.46,324.60,0.00),v40,fine,tPen\WObj:=wPaper;
    MoveL Offs(pOrigin,254.46,324.60,6.00),v60,z5,tPen\WObj:=wPaper;
    MoveL Offs(pOrigin,254.25,323.35,6.00),vTravel,z5,tPen\WObj:=wPaper;
    MoveL Offs(pOrigin,254.25,323.35,0.00),v60,z0,tPen\WObj:=wPaper;
    MoveL Offs(pOrigin,258.71,323.35,0.00),v40,z0,tPen\WObj:=wPaper;
    MoveL Offs(pOrigin,259.06,323.57,0.00),v40,z0,tPen\WObj:=wPaper;
    MoveL Offs(pOrigin,249.29,313.80,0.00),v40,z0,tPen\WObj:=wPaper;
    MoveL Offs(pOrigin,249.36,312.70,0.00),v40,z0,tPen\WObj:=wPaper;
    MoveL Offs(pOrigin,248.94,313.12,0.00),v40,z0,tPen\WObj:=wPaper;
    MoveL Offs(pOrigin,248.94,315.04,0.00),v40,z0,tPen\WObj:=wPaper;
    MoveL Offs(pOrigin,249.36,316.74,0.00),v40,fine,tPen\WObj:=wPaper;
    MoveL Offs(pOrigin,249.36,316.74,6.00),v60,z5,tPen\WObj:=wPaper;
    MoveL Offs(pOrigin,248.30,316.10,6.00),vTravel,z5,tPen\WObj:=wPaper;
    MoveL Offs(pOrigin,248.30,316.10,0.00),v60,z0,tPen\WObj:=wPaper;
    MoveL Offs(pOrigin,248.73,316.52,0.00),v40,z0,tPen\WObj:=wPaper;
    MoveL Offs(pOrigin,248.30,316.10,0.00),v40,fine,tPen\WObj:=wPaper;
    MoveL Offs(pOrigin,248.30,316.10,6.00),v60,z5,tPen\WObj:=wPaper;
    MoveL Offs(pOrigin,247.45,317.02,6.00),vTravel,z5,tPen\WObj:=wPaper;
    MoveL Offs(pOrigin,247.45,317.02,0.00),v60,z0,tPen\WObj:=wPaper;
    MoveL Offs(pOrigin,272.74,317.02,0.00),v40,z0,tPen\WObj:=wPaper;
    MoveL Offs(pOrigin,272.74,318.07,0.00),v40,z0,tPen\WObj:=wPaper;
    MoveL Offs(pOrigin,268.91,318.07,0.00),v40,z0,tPen\WObj:=wPaper;
    MoveL Offs(pOrigin,269.29,317.59,0.00),v40,z0,tPen\WObj:=wPaper;
    MoveL Offs(pOrigin,269.29,314.40,0.00),v40,z0,tPen\WObj:=wPaper;
    MoveL Offs(pOrigin,269.76,313.55,0.00),v40,z0,tPen\WObj:=wPaper;
    MoveL Offs(pOrigin,269.34,313.98,0.00),v40,z0,tPen\WObj:=wPaper;
    MoveL Offs(pOrigin,268.27,313.98,0.00),v40,z0,tPen\WObj:=wPaper;
    MoveL Offs(pOrigin,268.27,313.98,0.00),v40,z0,tPen\WObj:=wPaper;
    MoveL Offs(pOrigin,268.20,312.91,0.00),v40,z0,tPen\WObj:=wPaper;
    MoveL Offs(pOrigin,268.49,312.70,0.00),v40,z0,tPen\WObj:=wPaper;
    MoveL Offs(pOrigin,269.12,312.77,0.00),v40,z0,tPen\WObj:=wPaper;
    MoveL Offs(pOrigin,270.61,313.76,0.00),v40,z0,tPen\WObj:=wPaper;
    MoveL Offs(pOrigin,271.04,313.85,0.00),v40,z0,tPen\WObj:=wPaper;
    MoveL Offs(pOrigin,258.08,313.85,0.00),v40,z0,tPen\WObj:=wPaper;
    MoveL Offs(pOrigin,258.50,312.79,0.00),v40,z0,tPen\WObj:=wPaper;
    MoveL Offs(pOrigin,257.44,312.79,0.00),v40,z0,tPen\WObj:=wPaper;
    MoveL Offs(pOrigin,258.12,312.18,0.00),v40,z0,tPen\WObj:=wPaper;
    MoveL Offs(pOrigin,267.14,321.19,0.00),v40,z0,tPen\WObj:=wPaper;
    MoveL Offs(pOrigin,267.00,320.99,0.00),v40,z0,tPen\WObj:=wPaper;
    MoveL Offs(pOrigin,267.42,320.56,0.00),v40,z0,tPen\WObj:=wPaper;
    MoveL Offs(pOrigin,268.49,320.35,0.00),v40,z0,tPen\WObj:=wPaper;
    MoveL Offs(pOrigin,268.49,320.35,0.00),v40,z0,tPen\WObj:=wPaper;
    MoveL Offs(pOrigin,272.52,323.54,0.00),v40,z0,tPen\WObj:=wPaper;
    MoveL Offs(pOrigin,273.16,324.46,0.00),v40,z0,tPen\WObj:=wPaper;
    MoveL Offs(pOrigin,275.71,325.45,0.00),v40,z0,tPen\WObj:=wPaper;
    MoveL Offs(pOrigin,277.20,325.66,0.00),v40,z0,tPen\WObj:=wPaper;
    MoveL Offs(pOrigin,279.33,325.45,0.00),v40,z0,tPen\WObj:=wPaper;
    MoveL Offs(pOrigin,280.17,325.73,0.00),v40,z0,tPen\WObj:=wPaper;
    MoveL Offs(pOrigin,284.64,323.89,0.00),v40,z0,tPen\WObj:=wPaper;
    MoveL Offs(pOrigin,285.06,322.69,0.00),v40,z0,tPen\WObj:=wPaper;
    MoveL Offs(pOrigin,285.06,322.69,0.00),v40,z0,tPen\WObj:=wPaper;
    MoveL Offs(pOrigin,283.58,322.90,0.00),v40,z0,tPen\WObj:=wPaper;
    MoveL Offs(pOrigin,283.58,322.90,0.00),v40,z0,tPen\WObj:=wPaper;
  ENDPROC

  PROC DrawPart122()
    MoveL Offs(pOrigin,283.36,324.17,0.00),v40,z0,tPen\WObj:=wPaper;
    MoveL Offs(pOrigin,283.79,324.41,0.00),v40,z0,tPen\WObj:=wPaper;
    MoveL Offs(pOrigin,279.32,324.41,0.00),v40,z0,tPen\WObj:=wPaper;
    MoveL Offs(pOrigin,279.13,324.23,0.00),v40,z0,tPen\WObj:=wPaper;
    MoveL Offs(pOrigin,281.54,326.63,0.00),v40,z0,tPen\WObj:=wPaper;
    MoveL Offs(pOrigin,282.58,326.19,0.00),v40,z0,tPen\WObj:=wPaper;
    MoveL Offs(pOrigin,279.88,323.48,0.00),v40,z0,tPen\WObj:=wPaper;
    MoveL Offs(pOrigin,280.78,322.88,0.00),v40,z0,tPen\WObj:=wPaper;
    MoveL Offs(pOrigin,283.33,325.44,0.00),v40,z0,tPen\WObj:=wPaper;
    MoveL Offs(pOrigin,283.30,326.26,0.00),v40,z0,tPen\WObj:=wPaper;
    MoveL Offs(pOrigin,288.86,320.70,0.00),v40,z0,tPen\WObj:=wPaper;
    MoveL Offs(pOrigin,288.41,320.06,0.00),v40,z0,tPen\WObj:=wPaper;
    MoveL Offs(pOrigin,286.45,318.11,0.00),v40,z0,tPen\WObj:=wPaper;
    MoveL Offs(pOrigin,286.34,318.23,0.00),v40,z0,tPen\WObj:=wPaper;
    MoveL Offs(pOrigin,286.76,318.01,0.00),v40,z0,tPen\WObj:=wPaper;
    MoveL Offs(pOrigin,284.85,319.29,0.00),v40,z0,tPen\WObj:=wPaper;
    MoveL Offs(pOrigin,284.85,319.29,0.00),v40,z0,tPen\WObj:=wPaper;
    MoveL Offs(pOrigin,284.85,320.28,0.00),v40,z0,tPen\WObj:=wPaper;
    MoveL Offs(pOrigin,282.51,321.41,0.00),v40,z0,tPen\WObj:=wPaper;
    MoveL Offs(pOrigin,279.96,321.70,0.00),v40,z0,tPen\WObj:=wPaper;
    MoveL Offs(pOrigin,279.75,322.26,0.00),v40,z0,tPen\WObj:=wPaper;
    MoveL Offs(pOrigin,279.75,322.26,0.00),v40,z0,tPen\WObj:=wPaper;
    MoveL Offs(pOrigin,277.62,321.77,0.00),v40,z0,tPen\WObj:=wPaper;
    MoveL Offs(pOrigin,277.20,321.06,0.00),v40,z0,tPen\WObj:=wPaper;
    MoveL Offs(pOrigin,275.71,320.35,0.00),v40,z0,tPen\WObj:=wPaper;
    MoveL Offs(pOrigin,275.71,320.35,0.00),v40,z0,tPen\WObj:=wPaper;
    MoveL Offs(pOrigin,272.95,319.08,0.00),v40,z0,tPen\WObj:=wPaper;
    MoveL Offs(pOrigin,272.10,319.15,0.00),v40,z0,tPen\WObj:=wPaper;
    MoveL Offs(pOrigin,271.89,319.50,0.00),v40,z0,tPen\WObj:=wPaper;
    MoveL Offs(pOrigin,271.89,319.50,0.00),v40,z0,tPen\WObj:=wPaper;
    MoveL Offs(pOrigin,272.17,320.07,0.00),v40,z0,tPen\WObj:=wPaper;
    MoveL Offs(pOrigin,274.01,321.20,0.00),v40,z0,tPen\WObj:=wPaper;
    MoveL Offs(pOrigin,274.18,320.44,0.00),v40,z0,tPen\WObj:=wPaper;
    MoveL Offs(pOrigin,277.19,317.44,0.00),v40,z0,tPen\WObj:=wPaper;
    MoveL Offs(pOrigin,276.14,317.59,0.00),v40,z0,tPen\WObj:=wPaper;
    MoveL Offs(pOrigin,277.62,317.87,0.00),v40,z0,tPen\WObj:=wPaper;
    MoveL Offs(pOrigin,279.96,319.43,0.00),v40,z0,tPen\WObj:=wPaper;
    MoveL Offs(pOrigin,281.66,319.71,0.00),v40,z0,tPen\WObj:=wPaper;
    MoveL Offs(pOrigin,281.66,319.71,0.00),v40,z0,tPen\WObj:=wPaper;
    MoveL Offs(pOrigin,282.09,320.35,0.00),v40,z0,tPen\WObj:=wPaper;
    MoveL Offs(pOrigin,283.58,320.35,0.00),v40,z0,tPen\WObj:=wPaper;
    MoveL Offs(pOrigin,283.58,320.56,0.00),v40,z0,tPen\WObj:=wPaper;
    MoveL Offs(pOrigin,283.02,320.64,0.00),v40,z0,tPen\WObj:=wPaper;
    MoveL Offs(pOrigin,286.02,323.65,0.00),v40,z0,tPen\WObj:=wPaper;
    MoveL Offs(pOrigin,285.91,323.96,0.00),v40,z0,tPen\WObj:=wPaper;
    MoveL Offs(pOrigin,285.49,324.39,0.00),v40,z0,tPen\WObj:=wPaper;
    MoveL Offs(pOrigin,285.91,323.96,0.00),v40,z0,tPen\WObj:=wPaper;
    MoveL Offs(pOrigin,285.27,324.40,0.00),v40,z0,tPen\WObj:=wPaper;
    MoveL Offs(pOrigin,282.27,321.39,0.00),v40,z0,tPen\WObj:=wPaper;
    MoveL Offs(pOrigin,282.73,322.30,0.00),v40,z0,tPen\WObj:=wPaper;
    MoveL Offs(pOrigin,286.12,322.30,0.00),v40,z0,tPen\WObj:=wPaper;
    MoveL Offs(pOrigin,285.91,321.62,0.00),v40,z0,tPen\WObj:=wPaper;
    MoveL Offs(pOrigin,285.06,322.69,0.00),v40,z0,tPen\WObj:=wPaper;
    MoveL Offs(pOrigin,285.27,323.35,0.00),v40,z0,tPen\WObj:=wPaper;
    MoveL Offs(pOrigin,281.45,323.35,0.00),v40,z0,tPen\WObj:=wPaper;
    MoveL Offs(pOrigin,281.88,322.69,0.00),v40,z0,tPen\WObj:=wPaper;
    MoveL Offs(pOrigin,283.36,322.48,0.00),v40,z0,tPen\WObj:=wPaper;
    MoveL Offs(pOrigin,283.58,322.90,0.00),v40,fine,tPen\WObj:=wPaper;
    MoveL Offs(pOrigin,283.58,322.90,6.00),v60,z5,tPen\WObj:=wPaper;
    MoveL Offs(pOrigin,283.58,321.24,6.00),vTravel,z5,tPen\WObj:=wPaper;
    MoveL Offs(pOrigin,283.58,321.24,0.00),v60,z0,tPen\WObj:=wPaper;
    MoveL Offs(pOrigin,286.76,321.24,0.00),v40,z0,tPen\WObj:=wPaper;
    MoveL Offs(pOrigin,286.34,321.41,0.00),v40,z0,tPen\WObj:=wPaper;
    MoveL Offs(pOrigin,287.61,320.00,0.00),v40,z0,tPen\WObj:=wPaper;
    MoveL Offs(pOrigin,288.46,319.71,0.00),v40,z0,tPen\WObj:=wPaper;
    MoveL Offs(pOrigin,288.25,319.13,0.00),v40,z0,tPen\WObj:=wPaper;
    MoveL Offs(pOrigin,285.70,319.13,0.00),v40,z0,tPen\WObj:=wPaper;
    MoveL Offs(pOrigin,285.56,318.70,0.00),v40,z0,tPen\WObj:=wPaper;
    MoveL Offs(pOrigin,287.96,321.11,0.00),v40,z0,tPen\WObj:=wPaper;
    MoveL Offs(pOrigin,287.61,322.05,0.00),v40,z0,tPen\WObj:=wPaper;
    MoveL Offs(pOrigin,287.19,322.48,0.00),v40,z0,tPen\WObj:=wPaper;
    MoveL Offs(pOrigin,287.61,322.05,0.00),v40,z0,tPen\WObj:=wPaper;
    MoveL Offs(pOrigin,287.36,322.01,0.00),v40,z0,tPen\WObj:=wPaper;
    MoveL Offs(pOrigin,284.66,319.30,0.00),v40,z0,tPen\WObj:=wPaper;
    MoveL Offs(pOrigin,284.85,319.29,0.00),v40,z0,tPen\WObj:=wPaper;
    MoveL Offs(pOrigin,281.66,319.71,0.00),v40,fine,tPen\WObj:=wPaper;
    MoveL Offs(pOrigin,281.66,319.71,6.00),v60,z5,tPen\WObj:=wPaper;
    MoveL Offs(pOrigin,283.03,319.07,6.00),vTravel,z5,tPen\WObj:=wPaper;
    MoveL Offs(pOrigin,283.03,319.07,0.00),v60,z0,tPen\WObj:=wPaper;
    MoveL Offs(pOrigin,265.75,336.35,0.00),v40,z0,tPen\WObj:=wPaper;
    MoveL Offs(pOrigin,265.54,336.02,0.00),v40,z0,tPen\WObj:=wPaper;
    MoveL Offs(pOrigin,263.13,333.62,0.00),v40,z0,tPen\WObj:=wPaper;
    MoveL Offs(pOrigin,263.81,333.91,0.00),v40,z0,tPen\WObj:=wPaper;
    MoveL Offs(pOrigin,268.06,333.91,0.00),v40,z0,tPen\WObj:=wPaper;
    MoveL Offs(pOrigin,268.38,334.38,0.00),v40,z0,tPen\WObj:=wPaper;
    MoveL Offs(pOrigin,265.67,331.68,0.00),v40,z0,tPen\WObj:=wPaper;
    MoveL Offs(pOrigin,265.73,332.25,0.00),v40,z0,tPen\WObj:=wPaper;
    MoveL Offs(pOrigin,266.36,329.49,0.00),v40,z0,tPen\WObj:=wPaper;
    MoveL Offs(pOrigin,266.15,327.58,0.00),v40,z0,tPen\WObj:=wPaper;
    MoveL Offs(pOrigin,265.37,325.45,0.00),v40,z0,tPen\WObj:=wPaper;
    MoveL Offs(pOrigin,264.02,323.54,0.00),v40,z0,tPen\WObj:=wPaper;
    MoveL Offs(pOrigin,262.75,323.11,0.00),v40,z0,tPen\WObj:=wPaper;
    MoveL Offs(pOrigin,262.75,323.11,0.00),v40,z0,tPen\WObj:=wPaper;
    MoveL Offs(pOrigin,264.24,327.79,0.00),v40,z0,tPen\WObj:=wPaper;
    MoveL Offs(pOrigin,264.02,330.34,0.00),v40,z0,tPen\WObj:=wPaper;
    MoveL Offs(pOrigin,263.39,331.61,0.00),v40,z0,tPen\WObj:=wPaper;
    MoveL Offs(pOrigin,263.39,331.61,0.00),v40,z0,tPen\WObj:=wPaper;
    MoveL Offs(pOrigin,263.39,332.25,0.00),v40,z0,tPen\WObj:=wPaper;
    MoveL Offs(pOrigin,262.54,332.67,0.00),v40,z0,tPen\WObj:=wPaper;
    MoveL Offs(pOrigin,262.54,332.67,0.00),v40,z0,tPen\WObj:=wPaper;
    MoveL Offs(pOrigin,262.11,334.16,0.00),v40,z0,tPen\WObj:=wPaper;
    MoveL Offs(pOrigin,262.11,334.16,0.00),v40,z0,tPen\WObj:=wPaper;
    MoveL Offs(pOrigin,263.39,334.02,0.00),v40,z0,tPen\WObj:=wPaper;
    MoveL Offs(pOrigin,265.09,332.25,0.00),v40,z0,tPen\WObj:=wPaper;
    MoveL Offs(pOrigin,265.08,332.57,0.00),v40,z0,tPen\WObj:=wPaper;
    MoveL Offs(pOrigin,267.48,334.98,0.00),v40,z0,tPen\WObj:=wPaper;
    MoveL Offs(pOrigin,267.18,334.16,0.00),v40,z0,tPen\WObj:=wPaper;
    MoveL Offs(pOrigin,267.18,331.82,0.00),v40,z0,tPen\WObj:=wPaper;
    MoveL Offs(pOrigin,266.36,331.80,0.00),v40,z0,tPen\WObj:=wPaper;
    MoveL Offs(pOrigin,269.55,331.80,0.00),v40,fine,tPen\WObj:=wPaper;
    MoveL Offs(pOrigin,269.55,331.80,6.00),v60,z5,tPen\WObj:=wPaper;
    MoveL Offs(pOrigin,268.70,332.86,6.00),vTravel,z5,tPen\WObj:=wPaper;
    MoveL Offs(pOrigin,268.70,332.86,0.00),v60,z0,tPen\WObj:=wPaper;
    MoveL Offs(pOrigin,265.30,332.86,0.00),v40,z0,tPen\WObj:=wPaper;
    MoveL Offs(pOrigin,265.07,333.52,0.00),v40,z0,tPen\WObj:=wPaper;
    MoveL Offs(pOrigin,265.07,335.01,0.00),v40,z0,tPen\WObj:=wPaper;
    MoveL Offs(pOrigin,264.01,335.44,0.00),v40,z0,tPen\WObj:=wPaper;
    MoveL Offs(pOrigin,264.01,334.38,0.00),v40,fine,tPen\WObj:=wPaper;
    MoveL Offs(pOrigin,264.01,334.38,6.00),v60,z5,tPen\WObj:=wPaper;
    MoveL Offs(pOrigin,264.18,333.17,6.00),vTravel,z5,tPen\WObj:=wPaper;
  ENDPROC

  PROC DrawPart123()
    MoveL Offs(pOrigin,264.18,333.17,0.00),v60,z0,tPen\WObj:=wPaper;
    MoveL Offs(pOrigin,266.58,335.57,0.00),v40,fine,tPen\WObj:=wPaper;
    MoveL Offs(pOrigin,266.58,335.57,6.00),v60,z5,tPen\WObj:=wPaper;
    MoveL Offs(pOrigin,264.49,336.47,6.00),vTravel,z5,tPen\WObj:=wPaper;
    MoveL Offs(pOrigin,264.49,336.47,0.00),v60,z0,tPen\WObj:=wPaper;
    MoveL Offs(pOrigin,262.08,334.06,0.00),v40,z0,tPen\WObj:=wPaper;
    MoveL Offs(pOrigin,261.19,334.66,0.00),v40,z0,tPen\WObj:=wPaper;
    MoveL Offs(pOrigin,263.14,336.61,0.00),v40,z0,tPen\WObj:=wPaper;
    MoveL Offs(pOrigin,263.81,336.02,0.00),v40,z0,tPen\WObj:=wPaper;
    MoveL Offs(pOrigin,260.41,336.02,0.00),v40,z0,tPen\WObj:=wPaper;
    MoveL Offs(pOrigin,260.29,335.25,0.00),v40,z0,tPen\WObj:=wPaper;
    MoveL Offs(pOrigin,262.09,337.06,0.00),v40,fine,tPen\WObj:=wPaper;
    MoveL Offs(pOrigin,262.09,337.06,6.00),v60,z5,tPen\WObj:=wPaper;
    MoveL Offs(pOrigin,259.55,337.50,6.00),vTravel,z5,tPen\WObj:=wPaper;
    MoveL Offs(pOrigin,259.55,337.50,0.00),v60,z0,tPen\WObj:=wPaper;
    MoveL Offs(pOrigin,255.79,333.74,0.00),v40,z0,tPen\WObj:=wPaper;
    MoveL Offs(pOrigin,256.80,333.91,0.00),v40,z0,tPen\WObj:=wPaper;
    MoveL Offs(pOrigin,258.71,333.91,0.00),v40,z0,tPen\WObj:=wPaper;
    MoveL Offs(pOrigin,259.09,334.05,0.00),v40,z0,tPen\WObj:=wPaper;
    MoveL Offs(pOrigin,257.29,332.25,0.00),v40,z0,tPen\WObj:=wPaper;
    MoveL Offs(pOrigin,257.65,332.86,0.00),v40,z0,tPen\WObj:=wPaper;
    MoveL Offs(pOrigin,259.14,332.86,0.00),v40,z0,tPen\WObj:=wPaper;
    MoveL Offs(pOrigin,259.53,333.01,0.00),v40,z0,tPen\WObj:=wPaper;
    MoveL Offs(pOrigin,257.73,331.20,0.00),v40,z0,tPen\WObj:=wPaper;
    MoveL Offs(pOrigin,258.29,331.80,0.00),v40,z0,tPen\WObj:=wPaper;
    MoveL Offs(pOrigin,259.56,331.80,0.00),v40,z0,tPen\WObj:=wPaper;
    MoveL Offs(pOrigin,259.98,331.96,0.00),v40,z0,tPen\WObj:=wPaper;
    MoveL Offs(pOrigin,258.18,330.15,0.00),v40,z0,tPen\WObj:=wPaper;
    MoveL Offs(pOrigin,258.50,330.74,0.00),v40,z0,tPen\WObj:=wPaper;
    MoveL Offs(pOrigin,259.77,330.74,0.00),v40,z0,tPen\WObj:=wPaper;
    MoveL Offs(pOrigin,260.43,330.91,0.00),v40,z0,tPen\WObj:=wPaper;
    MoveL Offs(pOrigin,258.17,328.66,0.00),v40,z0,tPen\WObj:=wPaper;
    MoveL Offs(pOrigin,258.71,329.69,0.00),v40,z0,tPen\WObj:=wPaper;
    MoveL Offs(pOrigin,259.77,329.69,0.00),v40,fine,tPen\WObj:=wPaper;
    MoveL Offs(pOrigin,259.77,329.69,6.00),v60,z5,tPen\WObj:=wPaper;
    MoveL Offs(pOrigin,260.97,330.67,6.00),vTravel,z5,tPen\WObj:=wPaper;
    MoveL Offs(pOrigin,260.97,330.67,0.00),v60,z0,tPen\WObj:=wPaper;
    MoveL Offs(pOrigin,251.80,339.84,0.00),v40,z0,tPen\WObj:=wPaper;
    MoveL Offs(pOrigin,251.70,339.19,0.00),v40,z0,tPen\WObj:=wPaper;
    MoveL Offs(pOrigin,248.51,339.19,0.00),v40,z0,tPen\WObj:=wPaper;
    MoveL Offs(pOrigin,248.17,339.56,0.00),v40,z0,tPen\WObj:=wPaper;
    MoveL Offs(pOrigin,242.76,334.15,0.00),v40,z0,tPen\WObj:=wPaper;
    MoveL Offs(pOrigin,242.77,333.95,0.00),v40,z0,tPen\WObj:=wPaper;
    MoveL Offs(pOrigin,242.99,333.52,0.00),v40,z0,tPen\WObj:=wPaper;
    MoveL Offs(pOrigin,242.77,333.95,0.00),v40,z0,tPen\WObj:=wPaper;
    MoveL Offs(pOrigin,242.14,334.59,0.00),v40,z0,tPen\WObj:=wPaper;
    MoveL Offs(pOrigin,242.35,334.16,0.00),v40,z0,tPen\WObj:=wPaper;
    MoveL Offs(pOrigin,242.14,334.59,0.00),v40,fine,tPen\WObj:=wPaper;
    MoveL Offs(pOrigin,242.14,334.59,6.00),v60,z5,tPen\WObj:=wPaper;
    MoveL Offs(pOrigin,241.50,335.65,6.00),vTravel,z5,tPen\WObj:=wPaper;
    MoveL Offs(pOrigin,241.50,335.65,0.00),v60,z0,tPen\WObj:=wPaper;
    MoveL Offs(pOrigin,242.00,334.59,0.00),v40,z0,tPen\WObj:=wPaper;
    MoveL Offs(pOrigin,243.91,332.46,0.00),v40,z0,tPen\WObj:=wPaper;
    MoveL Offs(pOrigin,244.26,331.40,0.00),v40,z0,tPen\WObj:=wPaper;
    MoveL Offs(pOrigin,244.05,328.21,0.00),v40,z0,tPen\WObj:=wPaper;
    MoveL Offs(pOrigin,244.05,328.21,0.00),v40,z0,tPen\WObj:=wPaper;
    MoveL Offs(pOrigin,244.26,328.00,0.00),v40,z0,tPen\WObj:=wPaper;
    MoveL Offs(pOrigin,244.05,326.94,0.00),v40,z0,tPen\WObj:=wPaper;
    MoveL Offs(pOrigin,244.05,326.94,0.00),v40,z0,tPen\WObj:=wPaper;
    MoveL Offs(pOrigin,243.41,327.15,0.00),v40,z0,tPen\WObj:=wPaper;
    MoveL Offs(pOrigin,243.41,327.58,0.00),v40,z0,tPen\WObj:=wPaper;
    MoveL Offs(pOrigin,244.05,328.21,0.00),v40,z0,tPen\WObj:=wPaper;
    MoveL Offs(pOrigin,243.60,328.63,0.00),v40,z0,tPen\WObj:=wPaper;
    MoveL Offs(pOrigin,262.98,309.24,0.00),v40,z0,tPen\WObj:=wPaper;
    MoveL Offs(pOrigin,263.36,309.95,0.00),v40,z0,tPen\WObj:=wPaper;
    MoveL Offs(pOrigin,272.52,319.11,0.00),v40,z0,tPen\WObj:=wPaper;
    MoveL Offs(pOrigin,271.89,319.50,0.00),v40,z0,tPen\WObj:=wPaper;
    MoveL Offs(pOrigin,270.40,318.86,0.00),v40,z0,tPen\WObj:=wPaper;
    MoveL Offs(pOrigin,268.91,318.86,0.00),v40,z0,tPen\WObj:=wPaper;
    MoveL Offs(pOrigin,267.21,318.23,0.00),v40,z0,tPen\WObj:=wPaper;
    MoveL Offs(pOrigin,266.36,318.44,0.00),v40,z0,tPen\WObj:=wPaper;
    MoveL Offs(pOrigin,264.88,317.80,0.00),v40,z0,tPen\WObj:=wPaper;
    MoveL Offs(pOrigin,264.88,317.80,0.00),v40,z0,tPen\WObj:=wPaper;
    MoveL Offs(pOrigin,264.02,317.59,0.00),v40,z0,tPen\WObj:=wPaper;
    MoveL Offs(pOrigin,263.81,317.80,0.00),v40,z0,tPen\WObj:=wPaper;
    MoveL Offs(pOrigin,264.24,318.07,0.00),v40,z0,tPen\WObj:=wPaper;
    MoveL Offs(pOrigin,235.76,318.07,0.00),v40,z0,tPen\WObj:=wPaper;
    MoveL Offs(pOrigin,236.56,318.44,0.00),v40,z0,tPen\WObj:=wPaper;
    MoveL Offs(pOrigin,236.56,317.16,0.00),v40,z0,tPen\WObj:=wPaper;
    MoveL Offs(pOrigin,235.55,317.02,0.00),v40,z0,tPen\WObj:=wPaper;
    MoveL Offs(pOrigin,237.68,317.02,0.00),v40,z0,tPen\WObj:=wPaper;
    MoveL Offs(pOrigin,237.68,316.95,0.00),v40,z0,tPen\WObj:=wPaper;
    MoveL Offs(pOrigin,237.25,314.83,0.00),v40,z0,tPen\WObj:=wPaper;
    MoveL Offs(pOrigin,237.46,312.49,0.00),v40,z0,tPen\WObj:=wPaper;
    MoveL Offs(pOrigin,237.25,312.06,0.00),v40,z0,tPen\WObj:=wPaper;
    MoveL Offs(pOrigin,237.25,312.06,0.00),v40,z0,tPen\WObj:=wPaper;
    MoveL Offs(pOrigin,236.68,312.49,0.00),v40,z0,tPen\WObj:=wPaper;
    MoveL Offs(pOrigin,236.33,314.19,0.00),v40,z0,tPen\WObj:=wPaper;
    MoveL Offs(pOrigin,235.98,314.40,0.00),v40,fine,tPen\WObj:=wPaper;
    MoveL Offs(pOrigin,235.98,314.40,6.00),v60,z5,tPen\WObj:=wPaper;
    MoveL Offs(pOrigin,234.61,314.05,6.00),vTravel,z5,tPen\WObj:=wPaper;
    MoveL Offs(pOrigin,234.61,314.05,0.00),v60,z0,tPen\WObj:=wPaper;
    MoveL Offs(pOrigin,246.93,326.38,0.00),v40,fine,tPen\WObj:=wPaper;
    MoveL Offs(pOrigin,246.93,326.38,6.00),v60,z5,tPen\WObj:=wPaper;
    MoveL Offs(pOrigin,247.80,327.41,6.00),vTravel,z5,tPen\WObj:=wPaper;
    MoveL Offs(pOrigin,247.80,327.41,0.00),v60,z0,tPen\WObj:=wPaper;
    MoveL Offs(pOrigin,243.74,331.47,0.00),v40,z0,tPen\WObj:=wPaper;
    MoveL Offs(pOrigin,244.70,331.61,0.00),v40,z0,tPen\WObj:=wPaper;
    MoveL Offs(pOrigin,246.05,332.96,0.00),v40,z0,tPen\WObj:=wPaper;
    MoveL Offs(pOrigin,245.61,334.01,0.00),v40,z0,tPen\WObj:=wPaper;
    MoveL Offs(pOrigin,244.10,332.51,0.00),v40,z0,tPen\WObj:=wPaper;
    MoveL Offs(pOrigin,243.41,333.10,0.00),v40,z0,tPen\WObj:=wPaper;
    MoveL Offs(pOrigin,243.62,332.67,0.00),v40,z0,tPen\WObj:=wPaper;
    MoveL Offs(pOrigin,243.41,333.10,0.00),v40,z0,tPen\WObj:=wPaper;
    MoveL Offs(pOrigin,243.36,333.26,0.00),v40,z0,tPen\WObj:=wPaper;
    MoveL Offs(pOrigin,246.81,336.71,0.00),v40,z0,tPen\WObj:=wPaper;
    MoveL Offs(pOrigin,246.60,336.71,0.00),v40,z0,tPen\WObj:=wPaper;
    MoveL Offs(pOrigin,244.26,337.77,0.00),v40,z0,tPen\WObj:=wPaper;
    MoveL Offs(pOrigin,244.05,338.41,0.00),v40,z0,tPen\WObj:=wPaper;
    MoveL Offs(pOrigin,244.05,338.41,0.00),v40,z0,tPen\WObj:=wPaper;
    MoveL Offs(pOrigin,245.32,338.62,0.00),v40,z0,tPen\WObj:=wPaper;
    MoveL Offs(pOrigin,245.32,338.62,0.00),v40,z0,tPen\WObj:=wPaper;
    MoveL Offs(pOrigin,245.32,338.84,0.00),v40,z0,tPen\WObj:=wPaper;
    MoveL Offs(pOrigin,246.39,338.62,0.00),v40,z0,tPen\WObj:=wPaper;
    MoveL Offs(pOrigin,246.39,337.99,0.00),v40,z0,tPen\WObj:=wPaper;
    MoveL Offs(pOrigin,245.75,337.99,0.00),v40,z0,tPen\WObj:=wPaper;
    MoveL Offs(pOrigin,245.32,338.62,0.00),v40,z0,tPen\WObj:=wPaper;
    MoveL Offs(pOrigin,245.32,339.70,0.00),v40,z0,tPen\WObj:=wPaper;
    MoveL Offs(pOrigin,241.27,335.65,0.00),v40,z0,tPen\WObj:=wPaper;
    MoveL Offs(pOrigin,241.50,335.65,0.00),v40,z0,tPen\WObj:=wPaper;
  ENDPROC

  PROC DrawPart124()
    MoveL Offs(pOrigin,237.25,337.21,0.00),v40,z0,tPen\WObj:=wPaper;
    MoveL Offs(pOrigin,236.40,338.41,0.00),v40,z0,tPen\WObj:=wPaper;
    MoveL Offs(pOrigin,236.48,338.33,0.00),v40,z0,tPen\WObj:=wPaper;
    MoveL Offs(pOrigin,237.98,339.83,0.00),v40,z0,tPen\WObj:=wPaper;
    MoveL Offs(pOrigin,238.17,340.03,0.00),v40,z0,tPen\WObj:=wPaper;
    MoveL Offs(pOrigin,247.79,330.41,0.00),v40,fine,tPen\WObj:=wPaper;
    MoveL Offs(pOrigin,247.79,330.41,6.00),v60,z5,tPen\WObj:=wPaper;
    MoveL Offs(pOrigin,249.29,330.41,6.00),vTravel,z5,tPen\WObj:=wPaper;
    MoveL Offs(pOrigin,249.29,330.41,0.00),v60,z0,tPen\WObj:=wPaper;
    MoveL Offs(pOrigin,299.47,280.22,0.00),v40,z0,tPen\WObj:=wPaper;
    MoveL Offs(pOrigin,299.07,279.95,0.00),v40,z0,tPen\WObj:=wPaper;
    MoveL Offs(pOrigin,284.79,265.67,0.00),v40,z0,tPen\WObj:=wPaper;
    MoveL Offs(pOrigin,284.09,265.74,0.00),v40,z0,tPen\WObj:=wPaper;
    MoveL Offs(pOrigin,295.36,254.47,0.00),v40,z0,tPen\WObj:=wPaper;
    MoveL Offs(pOrigin,294.35,254.32,0.00),v40,z0,tPen\WObj:=wPaper;
    MoveL Offs(pOrigin,290.14,250.11,0.00),v40,z0,tPen\WObj:=wPaper;
    MoveL Offs(pOrigin,290.16,250.65,0.00),v40,z0,tPen\WObj:=wPaper;
    MoveL Offs(pOrigin,289.95,251.50,0.00),v40,z0,tPen\WObj:=wPaper;
    MoveL Offs(pOrigin,290.80,251.71,0.00),v40,z0,tPen\WObj:=wPaper;
    MoveL Offs(pOrigin,290.14,251.61,0.00),v40,z0,tPen\WObj:=wPaper;
    MoveL Offs(pOrigin,293.75,255.21,0.00),v40,z0,tPen\WObj:=wPaper;
    MoveL Offs(pOrigin,293.00,255.96,0.00),v40,z0,tPen\WObj:=wPaper;
    MoveL Offs(pOrigin,291.65,254.61,0.00),v40,z0,tPen\WObj:=wPaper;
    MoveL Offs(pOrigin,291.01,254.33,0.00),v40,z0,tPen\WObj:=wPaper;
    MoveL Offs(pOrigin,293.72,251.63,0.00),v40,z0,tPen\WObj:=wPaper;
    MoveL Offs(pOrigin,294.46,252.37,0.00),v40,z0,tPen\WObj:=wPaper;
    MoveL Offs(pOrigin,291.16,255.68,0.00),v40,z0,tPen\WObj:=wPaper;
    MoveL Offs(pOrigin,291.66,256.11,0.00),v40,z0,tPen\WObj:=wPaper;
    MoveL Offs(pOrigin,292.56,257.01,0.00),v40,fine,tPen\WObj:=wPaper;
    MoveL Offs(pOrigin,292.56,257.01,6.00),v60,z5,tPen\WObj:=wPaper;
    MoveL Offs(pOrigin,292.26,258.21,6.00),vTravel,z5,tPen\WObj:=wPaper;
    MoveL Offs(pOrigin,292.26,258.21,0.00),v60,z0,tPen\WObj:=wPaper;
    MoveL Offs(pOrigin,291.36,257.30,0.00),v40,z0,tPen\WObj:=wPaper;
    MoveL Offs(pOrigin,291.65,258.09,0.00),v40,z0,tPen\WObj:=wPaper;
    MoveL Offs(pOrigin,292.71,257.66,0.00),v40,z0,tPen\WObj:=wPaper;
    MoveL Offs(pOrigin,293.14,253.41,0.00),v40,z0,tPen\WObj:=wPaper;
    MoveL Offs(pOrigin,293.14,253.41,0.00),v40,z0,tPen\WObj:=wPaper;
    MoveL Offs(pOrigin,292.50,251.71,0.00),v40,z0,tPen\WObj:=wPaper;
    MoveL Offs(pOrigin,291.15,249.80,0.00),v40,z0,tPen\WObj:=wPaper;
    MoveL Offs(pOrigin,290.38,249.38,0.00),v40,z0,tPen\WObj:=wPaper;
    MoveL Offs(pOrigin,289.38,249.99,0.00),v40,z0,tPen\WObj:=wPaper;
    MoveL Offs(pOrigin,291.03,248.34,0.00),v40,z0,tPen\WObj:=wPaper;
    MoveL Offs(pOrigin,291.63,249.23,0.00),v40,z0,tPen\WObj:=wPaper;
    MoveL Offs(pOrigin,289.52,251.34,0.00),v40,z0,tPen\WObj:=wPaper;
    MoveL Offs(pOrigin,289.95,251.71,0.00),v40,z0,tPen\WObj:=wPaper;
    MoveL Offs(pOrigin,289.52,255.11,0.00),v40,fine,tPen\WObj:=wPaper;
    MoveL Offs(pOrigin,289.52,255.11,6.00),v60,z5,tPen\WObj:=wPaper;
    MoveL Offs(pOrigin,290.42,253.43,6.00),vTravel,z5,tPen\WObj:=wPaper;
    MoveL Offs(pOrigin,290.42,253.43,0.00),v60,z0,tPen\WObj:=wPaper;
    MoveL Offs(pOrigin,292.97,250.88,0.00),v40,z0,tPen\WObj:=wPaper;
    MoveL Offs(pOrigin,292.22,250.13,0.00),v40,z0,tPen\WObj:=wPaper;
    MoveL Offs(pOrigin,289.82,252.54,0.00),v40,fine,tPen\WObj:=wPaper;
    MoveL Offs(pOrigin,289.82,252.54,6.00),v60,z5,tPen\WObj:=wPaper;
    MoveL Offs(pOrigin,291.86,252.60,6.00),vTravel,z5,tPen\WObj:=wPaper;
    MoveL Offs(pOrigin,291.86,252.60,0.00),v60,z0,tPen\WObj:=wPaper;
    MoveL Offs(pOrigin,292.92,252.60,0.00),v40,z0,tPen\WObj:=wPaper;
    MoveL Offs(pOrigin,293.14,253.41,0.00),v40,z0,tPen\WObj:=wPaper;
    MoveL Offs(pOrigin,293.77,253.48,0.00),v40,z0,tPen\WObj:=wPaper;
    MoveL Offs(pOrigin,294.27,254.26,0.00),v40,z0,tPen\WObj:=wPaper;
    MoveL Offs(pOrigin,294.84,257.88,0.00),v40,z0,tPen\WObj:=wPaper;
    MoveL Offs(pOrigin,294.30,257.02,0.00),v40,z0,tPen\WObj:=wPaper;
    MoveL Offs(pOrigin,295.50,255.81,0.00),v40,fine,tPen\WObj:=wPaper;
    MoveL Offs(pOrigin,295.50,255.81,6.00),v60,z5,tPen\WObj:=wPaper;
    MoveL Offs(pOrigin,293.40,257.92,6.00),vTravel,z5,tPen\WObj:=wPaper;
    MoveL Offs(pOrigin,293.40,257.92,0.00),v60,z0,tPen\WObj:=wPaper;
    MoveL Offs(pOrigin,283.48,267.83,0.00),v40,z0,tPen\WObj:=wPaper;
    MoveL Offs(pOrigin,284.05,267.92,0.00),v40,z0,tPen\WObj:=wPaper;
    MoveL Offs(pOrigin,298.63,282.49,0.00),v40,z0,tPen\WObj:=wPaper;
    MoveL Offs(pOrigin,298.24,282.17,0.00),v40,z0,tPen\WObj:=wPaper;
    MoveL Offs(pOrigin,290.80,282.17,0.00),v40,fine,tPen\WObj:=wPaper;
    MoveL Offs(pOrigin,290.80,282.17,6.00),v60,z5,tPen\WObj:=wPaper;
    MoveL Offs(pOrigin,289.52,284.28,6.00),vTravel,z5,tPen\WObj:=wPaper;
    MoveL Offs(pOrigin,289.52,284.28,0.00),v60,z0,tPen\WObj:=wPaper;
    MoveL Offs(pOrigin,287.61,284.28,0.00),v40,fine,tPen\WObj:=wPaper;
    MoveL Offs(pOrigin,287.61,284.28,6.00),v60,z5,tPen\WObj:=wPaper;
    MoveL Offs(pOrigin,286.34,284.44,6.00),vTravel,z5,tPen\WObj:=wPaper;
    MoveL Offs(pOrigin,286.34,284.44,0.00),v60,z0,tPen\WObj:=wPaper;
    MoveL Offs(pOrigin,284.85,284.65,0.00),v40,z0,tPen\WObj:=wPaper;
    MoveL Offs(pOrigin,284.85,284.65,0.00),v40,z0,tPen\WObj:=wPaper;
    MoveL Offs(pOrigin,285.35,283.02,0.00),v40,z0,tPen\WObj:=wPaper;
    MoveL Offs(pOrigin,290.16,280.40,0.00),v40,z0,tPen\WObj:=wPaper;
    MoveL Offs(pOrigin,291.65,280.40,0.00),v40,z0,tPen\WObj:=wPaper;
    MoveL Offs(pOrigin,294.41,281.46,0.00),v40,z0,tPen\WObj:=wPaper;
    MoveL Offs(pOrigin,295.26,281.46,0.00),v40,z0,tPen\WObj:=wPaper;
    MoveL Offs(pOrigin,294.64,282.31,0.00),v40,z0,tPen\WObj:=wPaper;
    MoveL Offs(pOrigin,294.64,283.59,0.00),v40,z0,tPen\WObj:=wPaper;
    MoveL Offs(pOrigin,293.77,283.22,0.00),v40,z0,tPen\WObj:=wPaper;
    MoveL Offs(pOrigin,298.24,283.22,0.00),v40,z0,tPen\WObj:=wPaper;
    MoveL Offs(pOrigin,298.45,283.38,0.00),v40,z0,tPen\WObj:=wPaper;
    MoveL Offs(pOrigin,298.02,282.95,0.00),v40,z0,tPen\WObj:=wPaper;
    MoveL Offs(pOrigin,298.02,282.10,0.00),v40,z0,tPen\WObj:=wPaper;
    MoveL Offs(pOrigin,298.45,281.67,0.00),v40,z0,tPen\WObj:=wPaper;
    MoveL Offs(pOrigin,299.09,281.67,0.00),v40,z0,tPen\WObj:=wPaper;
    MoveL Offs(pOrigin,299.47,281.72,0.00),v40,z0,tPen\WObj:=wPaper;
    MoveL Offs(pOrigin,241.17,340.02,0.00),v40,z0,tPen\WObj:=wPaper;
    MoveL Offs(pOrigin,240.83,339.69,0.00),v40,z0,tPen\WObj:=wPaper;
    MoveL Offs(pOrigin,238.28,337.13,0.00),v40,z0,tPen\WObj:=wPaper;
    MoveL Offs(pOrigin,237.38,337.73,0.00),v40,z0,tPen\WObj:=wPaper;
    MoveL Offs(pOrigin,239.48,339.83,0.00),v40,z0,tPen\WObj:=wPaper;
    MoveL Offs(pOrigin,239.67,340.02,0.00),v40,z0,tPen\WObj:=wPaper;
    MoveL Offs(pOrigin,247.18,332.51,0.00),v40,fine,tPen\WObj:=wPaper;
    MoveL Offs(pOrigin,247.18,332.51,6.00),v60,z5,tPen\WObj:=wPaper;
    MoveL Offs(pOrigin,247.41,334.32,6.00),vTravel,z5,tPen\WObj:=wPaper;
    MoveL Offs(pOrigin,247.41,334.32,0.00),v60,z0,tPen\WObj:=wPaper;
    MoveL Offs(pOrigin,248.61,335.52,0.00),v40,z0,tPen\WObj:=wPaper;
    MoveL Offs(pOrigin,248.72,334.97,0.00),v40,z0,tPen\WObj:=wPaper;
    MoveL Offs(pOrigin,247.24,334.97,0.00),v40,z0,tPen\WObj:=wPaper;
    MoveL Offs(pOrigin,247.02,334.59,0.00),v40,z0,tPen\WObj:=wPaper;
    MoveL Offs(pOrigin,246.81,335.01,0.00),v40,z0,tPen\WObj:=wPaper;
    MoveL Offs(pOrigin,247.02,334.59,0.00),v40,z0,tPen\WObj:=wPaper;
    MoveL Offs(pOrigin,246.51,334.91,0.00),v40,z0,tPen\WObj:=wPaper;
    MoveL Offs(pOrigin,247.71,336.11,0.00),v40,z0,tPen\WObj:=wPaper;
    MoveL Offs(pOrigin,247.66,336.29,0.00),v40,z0,tPen\WObj:=wPaper;
    MoveL Offs(pOrigin,248.09,336.08,0.00),v40,z0,tPen\WObj:=wPaper;
    MoveL Offs(pOrigin,247.66,336.29,0.00),v40,fine,tPen\WObj:=wPaper;
    MoveL Offs(pOrigin,247.66,336.29,6.00),v60,z5,tPen\WObj:=wPaper;
    MoveL Offs(pOrigin,248.67,337.00,6.00),vTravel,z5,tPen\WObj:=wPaper;
    MoveL Offs(pOrigin,248.67,337.00,0.00),v60,z0,tPen\WObj:=wPaper;
    MoveL Offs(pOrigin,245.66,340.00,0.00),v40,fine,tPen\WObj:=wPaper;
    MoveL Offs(pOrigin,245.66,340.00,6.00),v60,z5,tPen\WObj:=wPaper;
  ENDPROC

  PROC DrawPart125()
    MoveL Offs(pOrigin,244.16,340.01,6.00),vTravel,z5,tPen\WObj:=wPaper;
    MoveL Offs(pOrigin,244.16,340.01,0.00),v60,z0,tPen\WObj:=wPaper;
    MoveL Offs(pOrigin,253.48,330.69,0.00),v40,z0,tPen\WObj:=wPaper;
    MoveL Offs(pOrigin,252.94,330.89,0.00),v40,z0,tPen\WObj:=wPaper;
    MoveL Offs(pOrigin,252.19,330.14,0.00),v40,fine,tPen\WObj:=wPaper;
    MoveL Offs(pOrigin,252.19,330.14,6.00),v60,z5,tPen\WObj:=wPaper;
    MoveL Offs(pOrigin,252.49,331.93,6.00),vTravel,z5,tPen\WObj:=wPaper;
    MoveL Offs(pOrigin,252.49,331.93,0.00),v60,z0,tPen\WObj:=wPaper;
    MoveL Offs(pOrigin,249.94,329.38,0.00),v40,z0,tPen\WObj:=wPaper;
    MoveL Offs(pOrigin,249.29,328.91,0.00),v40,z0,tPen\WObj:=wPaper;
    MoveL Offs(pOrigin,300.08,278.12,0.00),v40,z0,tPen\WObj:=wPaper;
    MoveL Offs(pOrigin,299.66,277.55,0.00),v40,z0,tPen\WObj:=wPaper;
    MoveL Offs(pOrigin,296.20,274.10,0.00),v40,z0,tPen\WObj:=wPaper;
    MoveL Offs(pOrigin,296.75,274.88,0.00),v40,z0,tPen\WObj:=wPaper;
    MoveL Offs(pOrigin,296.75,276.58,0.00),v40,fine,tPen\WObj:=wPaper;
    MoveL Offs(pOrigin,296.75,276.58,6.00),v60,z5,tPen\WObj:=wPaper;
    MoveL Offs(pOrigin,298.86,276.36,6.00),vTravel,z5,tPen\WObj:=wPaper;
    MoveL Offs(pOrigin,298.86,276.36,0.00),v60,z0,tPen\WObj:=wPaper;
    MoveL Offs(pOrigin,298.86,274.24,0.00),v40,z0,tPen\WObj:=wPaper;
    MoveL Offs(pOrigin,298.24,273.72,0.00),v40,z0,tPen\WObj:=wPaper;
    MoveL Offs(pOrigin,299.73,273.72,0.00),v40,z0,tPen\WObj:=wPaper;
    MoveL Offs(pOrigin,300.25,273.66,0.00),v40,z0,tPen\WObj:=wPaper;
    MoveL Offs(pOrigin,299.20,272.61,0.00),v40,z0,tPen\WObj:=wPaper;
    MoveL Offs(pOrigin,299.09,272.54,0.00),v40,z0,tPen\WObj:=wPaper;
    MoveL Offs(pOrigin,298.24,273.39,0.00),v40,z0,tPen\WObj:=wPaper;
    MoveL Offs(pOrigin,299.09,272.54,0.00),v40,z0,tPen\WObj:=wPaper;
    MoveL Offs(pOrigin,298.30,273.20,0.00),v40,z0,tPen\WObj:=wPaper;
    MoveL Offs(pOrigin,300.10,275.01,0.00),v40,z0,tPen\WObj:=wPaper;
    MoveL Offs(pOrigin,300.15,274.66,0.00),v40,z0,tPen\WObj:=wPaper;
    MoveL Offs(pOrigin,300.22,273.60,0.00),v40,z0,tPen\WObj:=wPaper;
    MoveL Offs(pOrigin,302.13,270.41,0.00),v40,z0,tPen\WObj:=wPaper;
    MoveL Offs(pOrigin,303.34,266.38,0.00),v40,z0,tPen\WObj:=wPaper;
    MoveL Offs(pOrigin,303.34,262.76,0.00),v40,z0,tPen\WObj:=wPaper;
    MoveL Offs(pOrigin,300.36,251.93,0.00),v40,z0,tPen\WObj:=wPaper;
    MoveL Offs(pOrigin,299.51,247.68,0.00),v40,z0,tPen\WObj:=wPaper;
    MoveL Offs(pOrigin,299.58,246.82,0.00),v40,z0,tPen\WObj:=wPaper;
    MoveL Offs(pOrigin,299.94,246.47,0.00),v40,z0,tPen\WObj:=wPaper;
    MoveL Offs(pOrigin,313.54,246.61,0.00),v40,z0,tPen\WObj:=wPaper;
    MoveL Offs(pOrigin,329.69,245.98,0.00),v40,z0,tPen\WObj:=wPaper;
    MoveL Offs(pOrigin,346.69,244.70,0.00),v40,z0,tPen\WObj:=wPaper;
    MoveL Offs(pOrigin,362.84,242.57,0.00),v40,z0,tPen\WObj:=wPaper;
    MoveL Offs(pOrigin,369.21,241.09,0.00),v40,z0,tPen\WObj:=wPaper;
    MoveL Offs(pOrigin,373.67,239.46,0.00),v40,z0,tPen\WObj:=wPaper;
    MoveL Offs(pOrigin,377.71,236.84,0.00),v40,z0,tPen\WObj:=wPaper;
    MoveL Offs(pOrigin,379.62,234.93,0.00),v40,z0,tPen\WObj:=wPaper;
    MoveL Offs(pOrigin,381.61,232.16,0.00),v40,z0,tPen\WObj:=wPaper;
    MoveL Offs(pOrigin,384.30,225.57,0.00),v40,z0,tPen\WObj:=wPaper;
    MoveL Offs(pOrigin,385.36,221.11,0.00),v40,z0,tPen\WObj:=wPaper;
    MoveL Offs(pOrigin,386.42,213.46,0.00),v40,z0,tPen\WObj:=wPaper;
    MoveL Offs(pOrigin,387.70,196.25,0.00),v40,z0,tPen\WObj:=wPaper;
    MoveL Offs(pOrigin,391.52,155.24,0.00),v40,z0,tPen\WObj:=wPaper;
    MoveL Offs(pOrigin,394.29,129.10,0.00),v40,z0,tPen\WObj:=wPaper;
    MoveL Offs(pOrigin,394.78,128.32,0.00),v40,z0,tPen\WObj:=wPaper;
    MoveL Offs(pOrigin,394.50,128.46,0.00),v40,z0,tPen\WObj:=wPaper;
    MoveL Offs(pOrigin,393.90,128.46,0.00),v40,z0,tPen\WObj:=wPaper;
    MoveL Offs(pOrigin,393.90,127.40,0.00),v40,z0,tPen\WObj:=wPaper;
    MoveL Offs(pOrigin,393.57,126.54,0.00),v40,z0,tPen\WObj:=wPaper;
    MoveL Offs(pOrigin,395.37,128.35,0.00),v40,z0,tPen\WObj:=wPaper;
    MoveL Offs(pOrigin,395.36,129.08,0.00),v40,z0,tPen\WObj:=wPaper;
    MoveL Offs(pOrigin,388.00,136.44,0.00),v40,z0,tPen\WObj:=wPaper;
    MoveL Offs(pOrigin,388.66,136.57,0.00),v40,z0,tPen\WObj:=wPaper;
    MoveL Offs(pOrigin,393.17,141.07,0.00),v40,z0,tPen\WObj:=wPaper;
    MoveL Offs(pOrigin,392.80,140.66,0.00),v40,z0,tPen\WObj:=wPaper;
    MoveL Offs(pOrigin,391.74,140.66,0.00),v40,z0,tPen\WObj:=wPaper;
    MoveL Offs(pOrigin,391.74,139.61,0.00),v40,z0,tPen\WObj:=wPaper;
    MoveL Offs(pOrigin,393.01,139.61,0.00),v40,z0,tPen\WObj:=wPaper;
    MoveL Offs(pOrigin,393.46,139.88,0.00),v40,z0,tPen\WObj:=wPaper;
    MoveL Offs(pOrigin,388.65,135.07,0.00),v40,z0,tPen\WObj:=wPaper;
    MoveL Offs(pOrigin,388.15,134.79,0.00),v40,z0,tPen\WObj:=wPaper;
    MoveL Offs(pOrigin,397.62,125.33,0.00),v40,z0,tPen\WObj:=wPaper;
    MoveL Offs(pOrigin,397.01,125.51,0.00),v40,z0,tPen\WObj:=wPaper;
    MoveL Offs(pOrigin,394.76,123.25,0.00),v40,z0,tPen\WObj:=wPaper;
    MoveL Offs(pOrigin,394.33,122.64,0.00),v40,z0,tPen\WObj:=wPaper;
    MoveL Offs(pOrigin,397.49,119.48,0.00),v40,z0,tPen\WObj:=wPaper;
    MoveL Offs(pOrigin,396.99,119.51,0.00),v40,z0,tPen\WObj:=wPaper;
    MoveL Offs(pOrigin,395.04,117.56,0.00),v40,z0,tPen\WObj:=wPaper;
    MoveL Offs(pOrigin,395.56,117.43,0.00),v40,z0,tPen\WObj:=wPaper;
    MoveL Offs(pOrigin,397.05,117.43,0.00),v40,z0,tPen\WObj:=wPaper;
    MoveL Offs(pOrigin,397.26,117.20,0.00),v40,z0,tPen\WObj:=wPaper;
    MoveL Offs(pOrigin,397.05,117.62,0.00),v40,z0,tPen\WObj:=wPaper;
    MoveL Offs(pOrigin,397.26,117.20,0.00),v40,z0,tPen\WObj:=wPaper;
    MoveL Offs(pOrigin,397.59,117.12,0.00),v40,z0,tPen\WObj:=wPaper;
    MoveL Offs(pOrigin,396.08,115.62,0.00),v40,z0,tPen\WObj:=wPaper;
    MoveL Offs(pOrigin,395.25,115.75,0.00),v40,z0,tPen\WObj:=wPaper;
    MoveL Offs(pOrigin,402.31,108.68,0.00),v40,z0,tPen\WObj:=wPaper;
    MoveL Offs(pOrigin,401.76,109.34,0.00),v40,z0,tPen\WObj:=wPaper;
    MoveL Offs(pOrigin,398.45,106.04,0.00),v40,z0,tPen\WObj:=wPaper;
    MoveL Offs(pOrigin,398.96,106.36,0.00),v40,z0,tPen\WObj:=wPaper;
    MoveL Offs(pOrigin,403.14,102.11,0.00),v40,z0,tPen\WObj:=wPaper;
    MoveL Offs(pOrigin,404.56,99.99,0.00),v40,z0,tPen\WObj:=wPaper;
    MoveL Offs(pOrigin,405.83,97.22,0.00),v40,z0,tPen\WObj:=wPaper;
    MoveL Offs(pOrigin,407.04,93.61,0.00),v40,z0,tPen\WObj:=wPaper;
    MoveL Offs(pOrigin,409.80,82.56,0.00),v40,z0,tPen\WObj:=wPaper;
    MoveL Offs(pOrigin,413.62,73.00,0.00),v40,z0,tPen\WObj:=wPaper;
    MoveL Offs(pOrigin,414.40,67.69,0.00),v40,z0,tPen\WObj:=wPaper;
    MoveL Offs(pOrigin,413.84,67.55,0.00),v40,z0,tPen\WObj:=wPaper;
    MoveL Offs(pOrigin,412.77,68.96,0.00),v40,z0,tPen\WObj:=wPaper;
    MoveL Offs(pOrigin,408.52,73.00,0.00),v40,z0,tPen\WObj:=wPaper;
    MoveL Offs(pOrigin,402.36,77.32,0.00),v40,z0,tPen\WObj:=wPaper;
    MoveL Offs(pOrigin,394.71,81.36,0.00),v40,z0,tPen\WObj:=wPaper;
    MoveL Offs(pOrigin,390.46,83.06,0.00),v40,z0,tPen\WObj:=wPaper;
    MoveL Offs(pOrigin,385.36,84.55,0.00),v40,z0,tPen\WObj:=wPaper;
    MoveL Offs(pOrigin,384.94,85.11,0.00),v40,fine,tPen\WObj:=wPaper;
    MoveL Offs(pOrigin,384.94,85.11,6.00),v60,z5,tPen\WObj:=wPaper;
    MoveL Offs(pOrigin,385.65,82.78,6.00),vTravel,z5,tPen\WObj:=wPaper;
    MoveL Offs(pOrigin,385.65,82.78,0.00),v60,z0,tPen\WObj:=wPaper;
    MoveL Offs(pOrigin,389.85,86.99,0.00),v40,fine,tPen\WObj:=wPaper;
    MoveL Offs(pOrigin,389.85,86.99,6.00),v60,z5,tPen\WObj:=wPaper;
    MoveL Offs(pOrigin,390.99,88.64,6.00),vTravel,z5,tPen\WObj:=wPaper;
    MoveL Offs(pOrigin,390.99,88.64,0.00),v60,z0,tPen\WObj:=wPaper;
    MoveL Offs(pOrigin,388.88,90.75,0.00),v40,z0,tPen\WObj:=wPaper;
    MoveL Offs(pOrigin,388.82,90.43,0.00),v40,z0,tPen\WObj:=wPaper;
    MoveL Offs(pOrigin,387.46,89.08,0.00),v40,z0,tPen\WObj:=wPaper;
    MoveL Offs(pOrigin,388.29,88.35,0.00),v40,z0,tPen\WObj:=wPaper;
    MoveL Offs(pOrigin,386.04,90.61,0.00),v40,fine,tPen\WObj:=wPaper;
    MoveL Offs(pOrigin,386.04,90.61,6.00),v60,z5,tPen\WObj:=wPaper;
    MoveL Offs(pOrigin,390.76,89.38,6.00),vTravel,z5,tPen\WObj:=wPaper;
    MoveL Offs(pOrigin,390.76,89.38,0.00),v60,z0,tPen\WObj:=wPaper;
    MoveL Offs(pOrigin,391.66,90.29,0.00),v40,fine,tPen\WObj:=wPaper;
    MoveL Offs(pOrigin,391.66,90.29,6.00),v60,z5,tPen\WObj:=wPaper;
  ENDPROC

  PROC DrawPart126()
    MoveL Offs(pOrigin,397.94,84.61,6.00),vTravel,z5,tPen\WObj:=wPaper;
    MoveL Offs(pOrigin,397.94,84.61,0.00),v60,z0,tPen\WObj:=wPaper;
    MoveL Offs(pOrigin,396.28,82.96,0.00),v40,fine,tPen\WObj:=wPaper;
    MoveL Offs(pOrigin,396.28,82.96,6.00),v60,z5,tPen\WObj:=wPaper;
    MoveL Offs(pOrigin,396.85,81.29,6.00),vTravel,z5,tPen\WObj:=wPaper;
    MoveL Offs(pOrigin,396.85,81.29,0.00),v60,z0,tPen\WObj:=wPaper;
    MoveL Offs(pOrigin,417.44,60.70,0.00),v40,fine,tPen\WObj:=wPaper;
    MoveL Offs(pOrigin,417.44,60.70,6.00),v60,z5,tPen\WObj:=wPaper;
    MoveL Offs(pOrigin,416.39,59.35,6.00),vTravel,z5,tPen\WObj:=wPaper;
    MoveL Offs(pOrigin,416.39,59.35,0.00),v60,z0,tPen\WObj:=wPaper;
    MoveL Offs(pOrigin,414.69,59.35,0.00),v40,z0,tPen\WObj:=wPaper;
    MoveL Offs(pOrigin,414.90,58.30,0.00),v40,z0,tPen\WObj:=wPaper;
    MoveL Offs(pOrigin,416.39,58.30,0.00),v40,z0,tPen\WObj:=wPaper;
    MoveL Offs(pOrigin,416.39,57.24,0.00),v40,z0,tPen\WObj:=wPaper;
    MoveL Offs(pOrigin,414.90,57.24,0.00),v40,z0,tPen\WObj:=wPaper;
    MoveL Offs(pOrigin,414.90,56.18,0.00),v40,z0,tPen\WObj:=wPaper;
    MoveL Offs(pOrigin,416.39,56.18,0.00),v40,fine,tPen\WObj:=wPaper;
    MoveL Offs(pOrigin,416.39,56.18,6.00),v60,z5,tPen\WObj:=wPaper;
    MoveL Offs(pOrigin,415.96,53.02,6.00),vTravel,z5,tPen\WObj:=wPaper;
    MoveL Offs(pOrigin,415.96,53.02,0.00),v60,z0,tPen\WObj:=wPaper;
    MoveL Offs(pOrigin,414.69,53.02,0.00),v40,z0,tPen\WObj:=wPaper;
    MoveL Offs(pOrigin,414.48,51.96,0.00),v40,z0,tPen\WObj:=wPaper;
    MoveL Offs(pOrigin,415.75,51.96,0.00),v40,z0,tPen\WObj:=wPaper;
    MoveL Offs(pOrigin,416.41,52.31,0.00),v40,z0,tPen\WObj:=wPaper;
    MoveL Offs(pOrigin,412.66,48.56,0.00),v40,z0,tPen\WObj:=wPaper;
    MoveL Offs(pOrigin,412.53,49.18,0.00),v40,z0,tPen\WObj:=wPaper;
    MoveL Offs(pOrigin,415.09,46.63,0.00),v40,z0,tPen\WObj:=wPaper;
    MoveL Offs(pOrigin,414.05,46.68,0.00),v40,z0,tPen\WObj:=wPaper;
    MoveL Offs(pOrigin,412.56,46.68,0.00),v40,z0,tPen\WObj:=wPaper;
    MoveL Offs(pOrigin,412.35,46.86,0.00),v40,z0,tPen\WObj:=wPaper;
    MoveL Offs(pOrigin,412.56,47.29,0.00),v40,z0,tPen\WObj:=wPaper;
    MoveL Offs(pOrigin,412.35,46.86,0.00),v40,fine,tPen\WObj:=wPaper;
    MoveL Offs(pOrigin,412.35,46.86,6.00),v60,z5,tPen\WObj:=wPaper;
    MoveL Offs(pOrigin,413.20,47.74,6.00),vTravel,z5,tPen\WObj:=wPaper;
    MoveL Offs(pOrigin,413.20,47.74,0.00),v60,z0,tPen\WObj:=wPaper;
    MoveL Offs(pOrigin,414.48,47.74,0.00),v40,z0,tPen\WObj:=wPaper;
    MoveL Offs(pOrigin,414.90,48.79,0.00),v40,z0,tPen\WObj:=wPaper;
    MoveL Offs(pOrigin,413.62,48.79,0.00),v40,z0,tPen\WObj:=wPaper;
    MoveL Offs(pOrigin,414.05,49.85,0.00),v40,z0,tPen\WObj:=wPaper;
    MoveL Offs(pOrigin,415.33,49.85,0.00),v40,z0,tPen\WObj:=wPaper;
    MoveL Offs(pOrigin,415.54,50.90,0.00),v40,z0,tPen\WObj:=wPaper;
    MoveL Offs(pOrigin,414.26,50.90,0.00),v40,z0,tPen\WObj:=wPaper;
    MoveL Offs(pOrigin,413.27,51.43,0.00),v40,z0,tPen\WObj:=wPaper;
    MoveL Offs(pOrigin,415.98,48.72,0.00),v40,fine,tPen\WObj:=wPaper;
    MoveL Offs(pOrigin,415.98,48.72,6.00),v60,z5,tPen\WObj:=wPaper;
    MoveL Offs(pOrigin,416.57,51.12,6.00),vTravel,z5,tPen\WObj:=wPaper;
    MoveL Offs(pOrigin,416.57,51.12,0.00),v60,z0,tPen\WObj:=wPaper;
    MoveL Offs(pOrigin,413.71,53.97,0.00),v40,fine,tPen\WObj:=wPaper;
    MoveL Offs(pOrigin,413.71,53.97,6.00),v60,z5,tPen\WObj:=wPaper;
    MoveL Offs(pOrigin,411.02,53.68,6.00),vTravel,z5,tPen\WObj:=wPaper;
    MoveL Offs(pOrigin,411.02,53.68,0.00),v60,z0,tPen\WObj:=wPaper;
    MoveL Offs(pOrigin,408.16,56.54,0.00),v40,z0,tPen\WObj:=wPaper;
    MoveL Offs(pOrigin,408.94,56.78,0.00),v40,z0,tPen\WObj:=wPaper;
    MoveL Offs(pOrigin,409.84,57.69,0.00),v40,z0,tPen\WObj:=wPaper;
    MoveL Offs(pOrigin,410.56,57.13,0.00),v40,z0,tPen\WObj:=wPaper;
    MoveL Offs(pOrigin,407.10,60.58,0.00),v40,z0,tPen\WObj:=wPaper;
    MoveL Offs(pOrigin,408.05,60.38,0.00),v40,z0,tPen\WObj:=wPaper;
    MoveL Offs(pOrigin,408.95,61.28,0.00),v40,z0,tPen\WObj:=wPaper;
    MoveL Offs(pOrigin,409.50,61.17,0.00),v40,z0,tPen\WObj:=wPaper;
    MoveL Offs(pOrigin,405.29,65.38,0.00),v40,z0,tPen\WObj:=wPaper;
    MoveL Offs(pOrigin,405.97,65.76,0.00),v40,z0,tPen\WObj:=wPaper;
    MoveL Offs(pOrigin,406.87,66.66,0.00),v40,z0,tPen\WObj:=wPaper;
    MoveL Offs(pOrigin,407.32,65.62,0.00),v40,z0,tPen\WObj:=wPaper;
    MoveL Offs(pOrigin,406.56,64.87,0.00),v40,z0,tPen\WObj:=wPaper;
    MoveL Offs(pOrigin,407.04,64.07,0.00),v40,z0,tPen\WObj:=wPaper;
    MoveL Offs(pOrigin,406.83,64.50,0.00),v40,z0,tPen\WObj:=wPaper;
    MoveL Offs(pOrigin,407.04,64.07,0.00),v40,z0,tPen\WObj:=wPaper;
    MoveL Offs(pOrigin,407.01,63.82,0.00),v40,z0,tPen\WObj:=wPaper;
    MoveL Offs(pOrigin,407.76,64.57,0.00),v40,z0,tPen\WObj:=wPaper;
    MoveL Offs(pOrigin,408.74,64.92,0.00),v40,z0,tPen\WObj:=wPaper;
    MoveL Offs(pOrigin,401.83,71.83,0.00),v40,fine,tPen\WObj:=wPaper;
    MoveL Offs(pOrigin,401.83,71.83,6.00),v60,z5,tPen\WObj:=wPaper;
    MoveL Offs(pOrigin,401.82,73.33,6.00),vTravel,z5,tPen\WObj:=wPaper;
    MoveL Offs(pOrigin,401.82,73.33,0.00),v60,z0,tPen\WObj:=wPaper;
    MoveL Offs(pOrigin,407.83,67.32,0.00),v40,fine,tPen\WObj:=wPaper;
    MoveL Offs(pOrigin,407.83,67.32,6.00),v60,z5,tPen\WObj:=wPaper;
    MoveL Offs(pOrigin,406.42,67.71,6.00),vTravel,z5,tPen\WObj:=wPaper;
    MoveL Offs(pOrigin,406.42,67.71,0.00),v60,z0,tPen\WObj:=wPaper;
    MoveL Offs(pOrigin,405.52,66.81,0.00),v40,z0,tPen\WObj:=wPaper;
    MoveL Offs(pOrigin,404.92,67.71,0.00),v40,z0,tPen\WObj:=wPaper;
    MoveL Offs(pOrigin,406.13,68.91,0.00),v40,z0,tPen\WObj:=wPaper;
    MoveL Offs(pOrigin,405.55,68.32,0.00),v40,z0,tPen\WObj:=wPaper;
    MoveL Offs(pOrigin,405.69,67.05,0.00),v40,z0,tPen\WObj:=wPaper;
    MoveL Offs(pOrigin,407.82,62.59,0.00),v40,z0,tPen\WObj:=wPaper;
    MoveL Offs(pOrigin,409.38,56.85,0.00),v40,z0,tPen\WObj:=wPaper;
    MoveL Offs(pOrigin,409.38,56.85,0.00),v40,z0,tPen\WObj:=wPaper;
    MoveL Offs(pOrigin,410.01,56.42,0.00),v40,z0,tPen\WObj:=wPaper;
    MoveL Offs(pOrigin,409.80,55.58,0.00),v40,z0,tPen\WObj:=wPaper;
    MoveL Offs(pOrigin,409.80,55.58,0.00),v40,z0,tPen\WObj:=wPaper;
    MoveL Offs(pOrigin,410.23,54.94,0.00),v40,z0,tPen\WObj:=wPaper;
    MoveL Offs(pOrigin,410.08,53.66,0.00),v40,z0,tPen\WObj:=wPaper;
    MoveL Offs(pOrigin,410.44,53.03,0.00),v40,z0,tPen\WObj:=wPaper;
    MoveL Offs(pOrigin,410.23,49.84,0.00),v40,z0,tPen\WObj:=wPaper;
    MoveL Offs(pOrigin,410.23,49.84,0.00),v40,z0,tPen\WObj:=wPaper;
    MoveL Offs(pOrigin,410.01,48.14,0.00),v40,z0,tPen\WObj:=wPaper;
    MoveL Offs(pOrigin,410.01,48.14,0.00),v40,z0,tPen\WObj:=wPaper;
    MoveL Offs(pOrigin,409.80,46.86,0.00),v40,z0,tPen\WObj:=wPaper;
    MoveL Offs(pOrigin,409.80,46.86,0.00),v40,z0,tPen\WObj:=wPaper;
    MoveL Offs(pOrigin,409.80,46.22,0.00),v40,z0,tPen\WObj:=wPaper;
    MoveL Offs(pOrigin,409.16,45.80,0.00),v40,z0,tPen\WObj:=wPaper;
    MoveL Offs(pOrigin,409.16,45.80,0.00),v40,z0,tPen\WObj:=wPaper;
    MoveL Offs(pOrigin,408.31,42.61,0.00),v40,z0,tPen\WObj:=wPaper;
    MoveL Offs(pOrigin,408.52,42.46,0.00),v40,z0,tPen\WObj:=wPaper;
    MoveL Offs(pOrigin,411.29,42.46,0.00),v40,z0,tPen\WObj:=wPaper;
    MoveL Offs(pOrigin,410.86,41.76,0.00),v40,z0,tPen\WObj:=wPaper;
    MoveL Offs(pOrigin,411.71,42.61,0.00),v40,z0,tPen\WObj:=wPaper;
    MoveL Offs(pOrigin,410.86,41.76,0.00),v40,z0,tPen\WObj:=wPaper;
    MoveL Offs(pOrigin,411.36,41.40,0.00),v40,z0,tPen\WObj:=wPaper;
    MoveL Offs(pOrigin,407.90,44.85,0.00),v40,z0,tPen\WObj:=wPaper;
    MoveL Offs(pOrigin,408.15,44.05,0.00),v40,z0,tPen\WObj:=wPaper;
    MoveL Offs(pOrigin,409.80,45.70,0.00),v40,z0,tPen\WObj:=wPaper;
    MoveL Offs(pOrigin,409.16,45.80,0.00),v40,z0,tPen\WObj:=wPaper;
    MoveL Offs(pOrigin,408.95,46.01,0.00),v40,z0,tPen\WObj:=wPaper;
    MoveL Offs(pOrigin,409.16,46.86,0.00),v40,z0,tPen\WObj:=wPaper;
    MoveL Offs(pOrigin,409.16,46.86,0.00),v40,z0,tPen\WObj:=wPaper;
    MoveL Offs(pOrigin,409.38,48.14,0.00),v40,z0,tPen\WObj:=wPaper;
    MoveL Offs(pOrigin,409.38,48.14,0.00),v40,z0,tPen\WObj:=wPaper;
    MoveL Offs(pOrigin,409.59,49.84,0.00),v40,z0,tPen\WObj:=wPaper;
    MoveL Offs(pOrigin,409.59,49.84,0.00),v40,z0,tPen\WObj:=wPaper;
    MoveL Offs(pOrigin,409.80,53.66,0.00),v40,z0,tPen\WObj:=wPaper;
  ENDPROC

  PROC DrawPart127()
    MoveL Offs(pOrigin,410.01,54.09,0.00),v40,z0,tPen\WObj:=wPaper;
    MoveL Offs(pOrigin,409.80,53.88,0.00),v40,z0,tPen\WObj:=wPaper;
    MoveL Offs(pOrigin,409.38,54.30,0.00),v40,z0,tPen\WObj:=wPaper;
    MoveL Offs(pOrigin,409.38,55.36,0.00),v40,z0,tPen\WObj:=wPaper;
    MoveL Offs(pOrigin,409.80,55.58,0.00),v40,z0,tPen\WObj:=wPaper;
    MoveL Offs(pOrigin,409.38,55.58,0.00),v40,z0,tPen\WObj:=wPaper;
    MoveL Offs(pOrigin,409.16,56.64,0.00),v40,z0,tPen\WObj:=wPaper;
    MoveL Offs(pOrigin,409.38,56.85,0.00),v40,z0,tPen\WObj:=wPaper;
    MoveL Offs(pOrigin,410.28,56.64,0.00),v40,z0,tPen\WObj:=wPaper;
    MoveL Offs(pOrigin,409.08,55.44,0.00),v40,z0,tPen\WObj:=wPaper;
    MoveL Offs(pOrigin,408.47,54.74,0.00),v40,z0,tPen\WObj:=wPaper;
    MoveL Offs(pOrigin,411.02,52.18,0.00),v40,z0,tPen\WObj:=wPaper;
    MoveL Offs(pOrigin,410.57,52.45,0.00),v40,z0,tPen\WObj:=wPaper;
    MoveL Offs(pOrigin,409.22,51.09,0.00),v40,z0,tPen\WObj:=wPaper;
    MoveL Offs(pOrigin,408.63,51.59,0.00),v40,z0,tPen\WObj:=wPaper;
    MoveL Offs(pOrigin,411.03,49.19,0.00),v40,z0,tPen\WObj:=wPaper;
    MoveL Offs(pOrigin,410.41,49.30,0.00),v40,z0,tPen\WObj:=wPaper;
    MoveL Offs(pOrigin,409.06,47.95,0.00),v40,z0,tPen\WObj:=wPaper;
    MoveL Offs(pOrigin,408.64,48.59,0.00),v40,z0,tPen\WObj:=wPaper;
    MoveL Offs(pOrigin,413.45,43.79,0.00),v40,z0,tPen\WObj:=wPaper;
    MoveL Offs(pOrigin,412.99,44.31,0.00),v40,z0,tPen\WObj:=wPaper;
    MoveL Offs(pOrigin,413.20,44.74,0.00),v40,z0,tPen\WObj:=wPaper;
    MoveL Offs(pOrigin,412.99,44.31,0.00),v40,z0,tPen\WObj:=wPaper;
    MoveL Offs(pOrigin,412.99,44.57,0.00),v40,z0,tPen\WObj:=wPaper;
    MoveL Offs(pOrigin,411.29,44.57,0.00),v40,z0,tPen\WObj:=wPaper;
    MoveL Offs(pOrigin,410.86,44.31,0.00),v40,z0,tPen\WObj:=wPaper;
    MoveL Offs(pOrigin,411.29,44.95,0.00),v40,z0,tPen\WObj:=wPaper;
    MoveL Offs(pOrigin,410.86,44.31,0.00),v40,z0,tPen\WObj:=wPaper;
    MoveL Offs(pOrigin,410.44,43.51,0.00),v40,z0,tPen\WObj:=wPaper;
    MoveL Offs(pOrigin,412.14,43.51,0.00),v40,z0,tPen\WObj:=wPaper;
    MoveL Offs(pOrigin,412.14,43.25,0.00),v40,z0,tPen\WObj:=wPaper;
    MoveL Offs(pOrigin,412.56,43.67,0.00),v40,z0,tPen\WObj:=wPaper;
    MoveL Offs(pOrigin,412.14,43.25,0.00),v40,z0,tPen\WObj:=wPaper;
    MoveL Offs(pOrigin,412.70,43.04,0.00),v40,z0,tPen\WObj:=wPaper;
    MoveL Offs(pOrigin,408.49,47.25,0.00),v40,z0,tPen\WObj:=wPaper;
    MoveL Offs(pOrigin,408.05,46.20,0.00),v40,z0,tPen\WObj:=wPaper;
    MoveL Offs(pOrigin,412.10,42.14,0.00),v40,fine,tPen\WObj:=wPaper;
    MoveL Offs(pOrigin,412.10,42.14,6.00),v60,z5,tPen\WObj:=wPaper;
    MoveL Offs(pOrigin,410.61,40.65,6.00),vTravel,z5,tPen\WObj:=wPaper;
    MoveL Offs(pOrigin,410.61,40.65,0.00),v60,z0,tPen\WObj:=wPaper;
    MoveL Offs(pOrigin,407.45,43.80,0.00),v40,z0,tPen\WObj:=wPaper;
    MoveL Offs(pOrigin,407.01,42.76,0.00),v40,z0,tPen\WObj:=wPaper;
    MoveL Offs(pOrigin,409.71,40.05,0.00),v40,z0,tPen\WObj:=wPaper;
    MoveL Offs(pOrigin,409.59,40.70,0.00),v40,z0,tPen\WObj:=wPaper;
    MoveL Offs(pOrigin,410.44,41.55,0.00),v40,z0,tPen\WObj:=wPaper;
    MoveL Offs(pOrigin,409.59,40.70,0.00),v40,z0,tPen\WObj:=wPaper;
    MoveL Offs(pOrigin,410.01,41.40,0.00),v40,z0,tPen\WObj:=wPaper;
    MoveL Offs(pOrigin,407.46,41.40,0.00),v40,z0,tPen\WObj:=wPaper;
    MoveL Offs(pOrigin,407.25,41.34,0.00),v40,z0,tPen\WObj:=wPaper;
    MoveL Offs(pOrigin,407.46,41.76,0.00),v40,z0,tPen\WObj:=wPaper;
    MoveL Offs(pOrigin,407.25,41.34,0.00),v40,z0,tPen\WObj:=wPaper;
    MoveL Offs(pOrigin,406.41,41.86,0.00),v40,z0,tPen\WObj:=wPaper;
    MoveL Offs(pOrigin,408.82,39.46,0.00),v40,z0,tPen\WObj:=wPaper;
    MoveL Offs(pOrigin,408.28,39.71,0.00),v40,z0,tPen\WObj:=wPaper;
    MoveL Offs(pOrigin,413.84,45.26,0.00),v40,z0,tPen\WObj:=wPaper;
    MoveL Offs(pOrigin,413.62,45.62,0.00),v40,z0,tPen\WObj:=wPaper;
    MoveL Offs(pOrigin,412.14,45.62,0.00),v40,fine,tPen\WObj:=wPaper;
    MoveL Offs(pOrigin,412.14,45.62,6.00),v60,z5,tPen\WObj:=wPaper;
    MoveL Offs(pOrigin,413.41,44.95,6.00),vTravel,z5,tPen\WObj:=wPaper;
    MoveL Offs(pOrigin,413.41,44.95,0.00),v60,z0,tPen\WObj:=wPaper;
    MoveL Offs(pOrigin,413.62,45.38,0.00),v40,z0,tPen\WObj:=wPaper;
    MoveL Offs(pOrigin,413.41,44.95,0.00),v40,z0,tPen\WObj:=wPaper;
    MoveL Offs(pOrigin,414.04,44.68,0.00),v40,z0,tPen\WObj:=wPaper;
    MoveL Offs(pOrigin,408.63,50.09,0.00),v40,z0,tPen\WObj:=wPaper;
    MoveL Offs(pOrigin,409.21,49.59,0.00),v40,z0,tPen\WObj:=wPaper;
    MoveL Offs(pOrigin,410.57,50.95,0.00),v40,z0,tPen\WObj:=wPaper;
    MoveL Offs(pOrigin,411.03,50.68,0.00),v40,z0,tPen\WObj:=wPaper;
    MoveL Offs(pOrigin,408.62,53.09,0.00),v40,z0,tPen\WObj:=wPaper;
    MoveL Offs(pOrigin,409.22,52.59,0.00),v40,z0,tPen\WObj:=wPaper;
    MoveL Offs(pOrigin,410.42,53.79,0.00),v40,fine,tPen\WObj:=wPaper;
    MoveL Offs(pOrigin,410.42,53.79,6.00),v60,z5,tPen\WObj:=wPaper;
    MoveL Offs(pOrigin,409.23,54.09,6.00),vTravel,z5,tPen\WObj:=wPaper;
    MoveL Offs(pOrigin,409.23,54.09,0.00),v60,z0,tPen\WObj:=wPaper;
    MoveL Offs(pOrigin,410.43,55.29,0.00),v40,z0,tPen\WObj:=wPaper;
    MoveL Offs(pOrigin,410.86,55.33,0.00),v40,z0,tPen\WObj:=wPaper;
    MoveL Offs(pOrigin,407.86,58.33,0.00),v40,z0,tPen\WObj:=wPaper;
    MoveL Offs(pOrigin,408.19,59.03,0.00),v40,z0,tPen\WObj:=wPaper;
    MoveL Offs(pOrigin,409.10,59.93,0.00),v40,z0,tPen\WObj:=wPaper;
    MoveL Offs(pOrigin,409.54,58.88,0.00),v40,z0,tPen\WObj:=wPaper;
    MoveL Offs(pOrigin,408.64,57.98,0.00),v40,fine,tPen\WObj:=wPaper;
    MoveL Offs(pOrigin,408.64,57.98,6.00),v60,z5,tPen\WObj:=wPaper;
    MoveL Offs(pOrigin,410.25,58.93,6.00),vTravel,z5,tPen\WObj:=wPaper;
    MoveL Offs(pOrigin,410.25,58.93,0.00),v60,z0,tPen\WObj:=wPaper;
    MoveL Offs(pOrigin,406.50,62.68,0.00),v40,z0,tPen\WObj:=wPaper;
    MoveL Offs(pOrigin,407.31,62.62,0.00),v40,z0,tPen\WObj:=wPaper;
    MoveL Offs(pOrigin,408.06,63.37,0.00),v40,z0,tPen\WObj:=wPaper;
    MoveL Offs(pOrigin,408.50,62.33,0.00),v40,z0,tPen\WObj:=wPaper;
    MoveL Offs(pOrigin,407.60,61.42,0.00),v40,fine,tPen\WObj:=wPaper;
    MoveL Offs(pOrigin,407.60,61.42,6.00),v60,z5,tPen\WObj:=wPaper;
    MoveL Offs(pOrigin,409.34,62.82,6.00),vTravel,z5,tPen\WObj:=wPaper;
    MoveL Offs(pOrigin,409.34,62.82,0.00),v60,z0,tPen\WObj:=wPaper;
    MoveL Offs(pOrigin,403.48,68.68,0.00),v40,z0,tPen\WObj:=wPaper;
    MoveL Offs(pOrigin,404.33,68.60,0.00),v40,z0,tPen\WObj:=wPaper;
    MoveL Offs(pOrigin,405.38,69.66,0.00),v40,z0,tPen\WObj:=wPaper;
    MoveL Offs(pOrigin,404.63,70.40,0.00),v40,z0,tPen\WObj:=wPaper;
    MoveL Offs(pOrigin,403.88,69.65,0.00),v40,fine,tPen\WObj:=wPaper;
    MoveL Offs(pOrigin,403.88,69.65,6.00),v60,z5,tPen\WObj:=wPaper;
    MoveL Offs(pOrigin,408.83,70.12,6.00),vTravel,z5,tPen\WObj:=wPaper;
    MoveL Offs(pOrigin,408.83,70.12,0.00),v60,z0,tPen\WObj:=wPaper;
    MoveL Offs(pOrigin,410.63,71.92,0.00),v40,fine,tPen\WObj:=wPaper;
    MoveL Offs(pOrigin,410.63,71.92,6.00),v60,z5,tPen\WObj:=wPaper;
    MoveL Offs(pOrigin,410.86,68.75,6.00),vTravel,z5,tPen\WObj:=wPaper;
    MoveL Offs(pOrigin,410.86,68.75,0.00),v60,z0,tPen\WObj:=wPaper;
    MoveL Offs(pOrigin,410.23,69.39,0.00),v40,z0,tPen\WObj:=wPaper;
    MoveL Offs(pOrigin,410.86,68.75,0.00),v40,fine,tPen\WObj:=wPaper;
    MoveL Offs(pOrigin,410.86,68.75,6.00),v60,z5,tPen\WObj:=wPaper;
    MoveL Offs(pOrigin,414.05,68.86,6.00),vTravel,z5,tPen\WObj:=wPaper;
    MoveL Offs(pOrigin,414.05,68.86,0.00),v60,z0,tPen\WObj:=wPaper;
    MoveL Offs(pOrigin,415.96,68.86,0.00),v40,z0,tPen\WObj:=wPaper;
    MoveL Offs(pOrigin,415.75,69.91,0.00),v40,z0,tPen\WObj:=wPaper;
    MoveL Offs(pOrigin,414.26,69.91,0.00),v40,fine,tPen\WObj:=wPaper;
    MoveL Offs(pOrigin,414.26,69.91,6.00),v60,z5,tPen\WObj:=wPaper;
    MoveL Offs(pOrigin,416.53,64.60,6.00),vTravel,z5,tPen\WObj:=wPaper;
    MoveL Offs(pOrigin,416.53,64.60,0.00),v60,z0,tPen\WObj:=wPaper;
    MoveL Offs(pOrigin,402.85,78.27,0.00),v40,z0,tPen\WObj:=wPaper;
    MoveL Offs(pOrigin,402.86,77.59,0.00),v40,z0,tPen\WObj:=wPaper;
    MoveL Offs(pOrigin,401.36,76.09,0.00),v40,z0,tPen\WObj:=wPaper;
    MoveL Offs(pOrigin,401.51,76.25,0.00),v40,z0,tPen\WObj:=wPaper;
    MoveL Offs(pOrigin,403.42,76.25,0.00),v40,fine,tPen\WObj:=wPaper;
    MoveL Offs(pOrigin,403.42,76.25,6.00),v60,z5,tPen\WObj:=wPaper;
  ENDPROC

  PROC DrawPart128()
    MoveL Offs(pOrigin,401.72,77.30,6.00),vTravel,z5,tPen\WObj:=wPaper;
    MoveL Offs(pOrigin,401.72,77.30,0.00),v60,z0,tPen\WObj:=wPaper;
    MoveL Offs(pOrigin,400.02,77.30,0.00),v40,z0,tPen\WObj:=wPaper;
    MoveL Offs(pOrigin,399.41,77.13,0.00),v40,z0,tPen\WObj:=wPaper;
    MoveL Offs(pOrigin,400.91,78.63,0.00),v40,z0,tPen\WObj:=wPaper;
    MoveL Offs(pOrigin,401.81,78.03,0.00),v40,z0,tPen\WObj:=wPaper;
    MoveL Offs(pOrigin,400.46,76.68,0.00),v40,fine,tPen\WObj:=wPaper;
    MoveL Offs(pOrigin,400.46,76.68,6.00),v60,z5,tPen\WObj:=wPaper;
    MoveL Offs(pOrigin,399.81,78.36,6.00),vTravel,z5,tPen\WObj:=wPaper;
    MoveL Offs(pOrigin,399.81,78.36,0.00),v60,z0,tPen\WObj:=wPaper;
    MoveL Offs(pOrigin,398.11,78.36,0.00),v40,z0,tPen\WObj:=wPaper;
    MoveL Offs(pOrigin,397.62,78.32,0.00),v40,z0,tPen\WObj:=wPaper;
    MoveL Offs(pOrigin,398.97,79.67,0.00),v40,z0,tPen\WObj:=wPaper;
    MoveL Offs(pOrigin,397.90,79.42,0.00),v40,z0,tPen\WObj:=wPaper;
    MoveL Offs(pOrigin,396.20,79.42,0.00),v40,z0,tPen\WObj:=wPaper;
    MoveL Offs(pOrigin,395.52,79.21,0.00),v40,z0,tPen\WObj:=wPaper;
    MoveL Offs(pOrigin,397.03,80.72,0.00),v40,z0,tPen\WObj:=wPaper;
    MoveL Offs(pOrigin,397.92,80.12,0.00),v40,z0,tPen\WObj:=wPaper;
    MoveL Offs(pOrigin,396.57,78.77,0.00),v40,fine,tPen\WObj:=wPaper;
    MoveL Offs(pOrigin,396.57,78.77,6.00),v60,z5,tPen\WObj:=wPaper;
    MoveL Offs(pOrigin,395.56,80.47,6.00),vTravel,z5,tPen\WObj:=wPaper;
    MoveL Offs(pOrigin,395.56,80.47,0.00),v60,z0,tPen\WObj:=wPaper;
    MoveL Offs(pOrigin,393.86,80.47,0.00),v40,z0,tPen\WObj:=wPaper;
    MoveL Offs(pOrigin,393.58,80.26,0.00),v40,z0,tPen\WObj:=wPaper;
    MoveL Offs(pOrigin,394.93,81.61,0.00),v40,z0,tPen\WObj:=wPaper;
    MoveL Offs(pOrigin,395.98,81.16,0.00),v40,z0,tPen\WObj:=wPaper;
    MoveL Offs(pOrigin,394.63,79.81,0.00),v40,fine,tPen\WObj:=wPaper;
    MoveL Offs(pOrigin,394.63,79.81,6.00),v60,z5,tPen\WObj:=wPaper;
    MoveL Offs(pOrigin,400.47,81.18,6.00),vTravel,z5,tPen\WObj:=wPaper;
    MoveL Offs(pOrigin,400.47,81.18,0.00),v60,z0,tPen\WObj:=wPaper;
    MoveL Offs(pOrigin,401.82,82.53,0.00),v40,fine,tPen\WObj:=wPaper;
    MoveL Offs(pOrigin,401.82,82.53,6.00),v60,z5,tPen\WObj:=wPaper;
    MoveL Offs(pOrigin,400.66,74.28,6.00),vTravel,z5,tPen\WObj:=wPaper;
    MoveL Offs(pOrigin,400.66,74.28,0.00),v60,z0,tPen\WObj:=wPaper;
    MoveL Offs(pOrigin,402.79,72.36,0.00),v40,z0,tPen\WObj:=wPaper;
    MoveL Offs(pOrigin,405.62,68.54,0.00),v40,z0,tPen\WObj:=wPaper;
    MoveL Offs(pOrigin,406.97,67.69,0.00),v40,z0,tPen\WObj:=wPaper;
    MoveL Offs(pOrigin,408.81,64.50,0.00),v40,z0,tPen\WObj:=wPaper;
    MoveL Offs(pOrigin,409.38,62.80,0.00),v40,fine,tPen\WObj:=wPaper;
    MoveL Offs(pOrigin,409.38,62.80,6.00),v60,z5,tPen\WObj:=wPaper;
    MoveL Offs(pOrigin,414.26,62.52,6.00),vTravel,z5,tPen\WObj:=wPaper;
    MoveL Offs(pOrigin,414.26,62.52,0.00),v60,z0,tPen\WObj:=wPaper;
    MoveL Offs(pOrigin,415.96,62.52,0.00),v40,fine,tPen\WObj:=wPaper;
    MoveL Offs(pOrigin,415.96,62.52,6.00),v60,z5,tPen\WObj:=wPaper;
    MoveL Offs(pOrigin,412.08,48.13,6.00),vTravel,z5,tPen\WObj:=wPaper;
    MoveL Offs(pOrigin,412.08,48.13,0.00),v60,z0,tPen\WObj:=wPaper;
    MoveL Offs(pOrigin,414.49,45.73,0.00),v40,z0,tPen\WObj:=wPaper;
    MoveL Offs(pOrigin,413.84,45.80,0.00),v40,z0,tPen\WObj:=wPaper;
    MoveL Offs(pOrigin,414.05,46.22,0.00),v40,z0,tPen\WObj:=wPaper;
    MoveL Offs(pOrigin,413.84,45.80,0.00),v40,fine,tPen\WObj:=wPaper;
    MoveL Offs(pOrigin,413.84,45.80,6.00),v60,z5,tPen\WObj:=wPaper;
    MoveL Offs(pOrigin,410.26,47.65,6.00),vTravel,z5,tPen\WObj:=wPaper;
    MoveL Offs(pOrigin,410.26,47.65,0.00),v60,z0,tPen\WObj:=wPaper;
    MoveL Offs(pOrigin,408.60,46.00,0.00),v40,fine,tPen\WObj:=wPaper;
    MoveL Offs(pOrigin,408.60,46.00,6.00),v60,z5,tPen\WObj:=wPaper;
    MoveL Offs(pOrigin,409.80,43.25,6.00),vTravel,z5,tPen\WObj:=wPaper;
    MoveL Offs(pOrigin,409.80,43.25,0.00),v60,z0,tPen\WObj:=wPaper;
    MoveL Offs(pOrigin,410.23,43.67,0.00),v40,z0,tPen\WObj:=wPaper;
    MoveL Offs(pOrigin,409.80,43.25,0.00),v40,fine,tPen\WObj:=wPaper;
    MoveL Offs(pOrigin,409.80,43.25,6.00),v60,z5,tPen\WObj:=wPaper;
    MoveL Offs(pOrigin,408.74,40.34,6.00),vTravel,z5,tPen\WObj:=wPaper;
    MoveL Offs(pOrigin,408.74,40.34,0.00),v60,z0,tPen\WObj:=wPaper;
    MoveL Offs(pOrigin,406.40,40.34,0.00),v40,z0,tPen\WObj:=wPaper;
    MoveL Offs(pOrigin,405.66,41.11,0.00),v40,z0,tPen\WObj:=wPaper;
    MoveL Offs(pOrigin,407.77,39.01,0.00),v40,z0,tPen\WObj:=wPaper;
    MoveL Offs(pOrigin,406.83,39.29,0.00),v40,z0,tPen\WObj:=wPaper;
    MoveL Offs(pOrigin,404.06,39.29,0.00),v40,z0,tPen\WObj:=wPaper;
    MoveL Offs(pOrigin,403.57,40.22,0.00),v40,z0,tPen\WObj:=wPaper;
    MoveL Offs(pOrigin,405.82,37.97,0.00),v40,z0,tPen\WObj:=wPaper;
    MoveL Offs(pOrigin,406.87,38.41,0.00),v40,z0,tPen\WObj:=wPaper;
    MoveL Offs(pOrigin,404.62,40.67,0.00),v40,z0,tPen\WObj:=wPaper;
    MoveL Offs(pOrigin,404.54,40.44,0.00),v40,z0,tPen\WObj:=wPaper;
    MoveL Offs(pOrigin,400.79,36.69,0.00),v40,z0,tPen\WObj:=wPaper;
    MoveL Offs(pOrigin,401.30,37.18,0.00),v40,z0,tPen\WObj:=wPaper;
    MoveL Offs(pOrigin,397.69,37.18,0.00),v40,z0,tPen\WObj:=wPaper;
    MoveL Offs(pOrigin,397.69,36.12,0.00),v40,z0,tPen\WObj:=wPaper;
    MoveL Offs(pOrigin,393.22,36.12,0.00),v40,fine,tPen\WObj:=wPaper;
    MoveL Offs(pOrigin,393.22,36.12,6.00),v60,z5,tPen\WObj:=wPaper;
    MoveL Offs(pOrigin,391.90,36.96,6.00),vTravel,z5,tPen\WObj:=wPaper;
    MoveL Offs(pOrigin,391.90,36.96,0.00),v60,z0,tPen\WObj:=wPaper;
    MoveL Offs(pOrigin,394.45,34.41,0.00),v40,fine,tPen\WObj:=wPaper;
    MoveL Offs(pOrigin,394.45,34.41,6.00),v60,z5,tPen\WObj:=wPaper;
    MoveL Offs(pOrigin,393.10,34.26,6.00),vTravel,z5,tPen\WObj:=wPaper;
    MoveL Offs(pOrigin,393.10,34.26,0.00),v60,z0,tPen\WObj:=wPaper;
    MoveL Offs(pOrigin,390.70,36.67,0.00),v40,z0,tPen\WObj:=wPaper;
    MoveL Offs(pOrigin,391.65,36.51,0.00),v40,z0,tPen\WObj:=wPaper;
    MoveL Offs(pOrigin,389.09,33.95,0.00),v40,z0,tPen\WObj:=wPaper;
    MoveL Offs(pOrigin,389.51,33.37,0.00),v40,z0,tPen\WObj:=wPaper;
    MoveL Offs(pOrigin,386.96,35.93,0.00),v40,z0,tPen\WObj:=wPaper;
    MoveL Offs(pOrigin,386.10,35.44,0.00),v40,z0,tPen\WObj:=wPaper;
    MoveL Offs(pOrigin,383.70,33.04,0.00),v40,z0,tPen\WObj:=wPaper;
    MoveL Offs(pOrigin,384.42,32.49,0.00),v40,z0,tPen\WObj:=wPaper;
    MoveL Offs(pOrigin,381.72,35.20,0.00),v40,fine,tPen\WObj:=wPaper;
    MoveL Offs(pOrigin,381.72,35.20,6.00),v60,z5,tPen\WObj:=wPaper;
    MoveL Offs(pOrigin,380.37,35.05,6.00),vTravel,z5,tPen\WObj:=wPaper;
    MoveL Offs(pOrigin,380.37,35.05,0.00),v60,z0,tPen\WObj:=wPaper;
    MoveL Offs(pOrigin,383.07,32.34,0.00),v40,z0,tPen\WObj:=wPaper;
    MoveL Offs(pOrigin,382.05,32.88,0.00),v40,z0,tPen\WObj:=wPaper;
    MoveL Offs(pOrigin,384.45,35.29,0.00),v40,z0,tPen\WObj:=wPaper;
    MoveL Offs(pOrigin,384.41,35.49,0.00),v40,z0,tPen\WObj:=wPaper;
    MoveL Offs(pOrigin,386.97,32.93,0.00),v40,fine,tPen\WObj:=wPaper;
    MoveL Offs(pOrigin,386.97,32.93,6.00),v60,z5,tPen\WObj:=wPaper;
    MoveL Offs(pOrigin,388.16,33.23,6.00),vTravel,z5,tPen\WObj:=wPaper;
    MoveL Offs(pOrigin,388.16,33.23,0.00),v60,z0,tPen\WObj:=wPaper;
    MoveL Offs(pOrigin,385.61,35.78,0.00),v40,fine,tPen\WObj:=wPaper;
    MoveL Offs(pOrigin,385.61,35.78,6.00),v60,z5,tPen\WObj:=wPaper;
    MoveL Offs(pOrigin,388.15,36.22,6.00),vTravel,z5,tPen\WObj:=wPaper;
    MoveL Offs(pOrigin,388.15,36.22,0.00),v60,z0,tPen\WObj:=wPaper;
    MoveL Offs(pOrigin,390.56,33.82,0.00),v40,fine,tPen\WObj:=wPaper;
    MoveL Offs(pOrigin,390.56,33.82,6.00),v60,z5,tPen\WObj:=wPaper;
    MoveL Offs(pOrigin,395.64,37.70,6.00),vTravel,z5,tPen\WObj:=wPaper;
    MoveL Offs(pOrigin,395.64,37.70,0.00),v60,z0,tPen\WObj:=wPaper;
    MoveL Offs(pOrigin,398.04,35.29,0.00),v40,fine,tPen\WObj:=wPaper;
    MoveL Offs(pOrigin,398.04,35.29,6.00),v60,z5,tPen\WObj:=wPaper;
    MoveL Offs(pOrigin,400.44,35.89,6.00),vTravel,z5,tPen\WObj:=wPaper;
    MoveL Offs(pOrigin,400.44,35.89,0.00),v60,z0,tPen\WObj:=wPaper;
    MoveL Offs(pOrigin,398.03,38.29,0.00),v40,z0,tPen\WObj:=wPaper;
    MoveL Offs(pOrigin,399.08,38.74,0.00),v40,z0,tPen\WObj:=wPaper;
    MoveL Offs(pOrigin,401.49,36.33,0.00),v40,fine,tPen\WObj:=wPaper;
    MoveL Offs(pOrigin,401.49,36.33,6.00),v60,z5,tPen\WObj:=wPaper;
  ENDPROC

  PROC DrawPart129()
    MoveL Offs(pOrigin,401.30,38.23,6.00),vTravel,z5,tPen\WObj:=wPaper;
    MoveL Offs(pOrigin,401.30,38.23,0.00),v60,z0,tPen\WObj:=wPaper;
    MoveL Offs(pOrigin,404.49,38.23,0.00),v40,fine,tPen\WObj:=wPaper;
    MoveL Offs(pOrigin,404.49,38.23,6.00),v60,z5,tPen\WObj:=wPaper;
    MoveL Offs(pOrigin,403.88,36.92,6.00),vTravel,z5,tPen\WObj:=wPaper;
    MoveL Offs(pOrigin,403.88,36.92,0.00),v60,z0,tPen\WObj:=wPaper;
    MoveL Offs(pOrigin,401.33,39.48,0.00),v40,fine,tPen\WObj:=wPaper;
    MoveL Offs(pOrigin,401.33,39.48,6.00),v60,z5,tPen\WObj:=wPaper;
    MoveL Offs(pOrigin,402.65,48.61,6.00),vTravel,z5,tPen\WObj:=wPaper;
    MoveL Offs(pOrigin,402.65,48.61,0.00),v60,z0,tPen\WObj:=wPaper;
    MoveL Offs(pOrigin,399.49,51.77,0.00),v40,fine,tPen\WObj:=wPaper;
    MoveL Offs(pOrigin,399.49,51.77,6.00),v60,z5,tPen\WObj:=wPaper;
    MoveL Offs(pOrigin,383.35,38.04,6.00),vTravel,z5,tPen\WObj:=wPaper;
    MoveL Offs(pOrigin,383.35,38.04,0.00),v60,z0,tPen\WObj:=wPaper;
    MoveL Offs(pOrigin,382.45,38.94,0.00),v40,fine,tPen\WObj:=wPaper;
    MoveL Offs(pOrigin,382.45,38.94,6.00),v60,z5,tPen\WObj:=wPaper;
    MoveL Offs(pOrigin,382.31,37.59,6.00),vTravel,z5,tPen\WObj:=wPaper;
    MoveL Offs(pOrigin,382.31,37.59,0.00),v60,z0,tPen\WObj:=wPaper;
    MoveL Offs(pOrigin,381.11,38.79,0.00),v40,fine,tPen\WObj:=wPaper;
    MoveL Offs(pOrigin,381.11,38.79,6.00),v60,z5,tPen\WObj:=wPaper;
    MoveL Offs(pOrigin,379.91,38.50,6.00),vTravel,z5,tPen\WObj:=wPaper;
    MoveL Offs(pOrigin,379.91,38.50,0.00),v60,z0,tPen\WObj:=wPaper;
    MoveL Offs(pOrigin,381.26,37.14,0.00),v40,fine,tPen\WObj:=wPaper;
    MoveL Offs(pOrigin,381.26,37.14,6.00),v60,z5,tPen\WObj:=wPaper;
    MoveL Offs(pOrigin,380.06,36.85,6.00),vTravel,z5,tPen\WObj:=wPaper;
    MoveL Offs(pOrigin,380.06,36.85,0.00),v60,z0,tPen\WObj:=wPaper;
    MoveL Offs(pOrigin,378.56,38.35,0.00),v40,fine,tPen\WObj:=wPaper;
    MoveL Offs(pOrigin,378.56,38.35,6.00),v60,z5,tPen\WObj:=wPaper;
    MoveL Offs(pOrigin,376.77,35.66,6.00),vTravel,z5,tPen\WObj:=wPaper;
    MoveL Offs(pOrigin,376.77,35.66,0.00),v60,z0,tPen\WObj:=wPaper;
    MoveL Offs(pOrigin,374.97,37.46,0.00),v40,fine,tPen\WObj:=wPaper;
    MoveL Offs(pOrigin,374.97,37.46,6.00),v60,z5,tPen\WObj:=wPaper;
    MoveL Offs(pOrigin,373.77,37.17,6.00),vTravel,z5,tPen\WObj:=wPaper;
    MoveL Offs(pOrigin,373.77,37.17,0.00),v60,z0,tPen\WObj:=wPaper;
    MoveL Offs(pOrigin,375.72,35.21,0.00),v40,fine,tPen\WObj:=wPaper;
    MoveL Offs(pOrigin,375.72,35.21,6.00),v60,z5,tPen\WObj:=wPaper;
    MoveL Offs(pOrigin,372.57,36.87,6.00),vTravel,z5,tPen\WObj:=wPaper;
    MoveL Offs(pOrigin,372.57,36.87,0.00),v60,z0,tPen\WObj:=wPaper;
    MoveL Offs(pOrigin,377.68,31.76,0.00),v40,fine,tPen\WObj:=wPaper;
    MoveL Offs(pOrigin,377.68,31.76,6.00),v60,z5,tPen\WObj:=wPaper;
    MoveL Offs(pOrigin,375.14,31.32,6.00),vTravel,z5,tPen\WObj:=wPaper;
    MoveL Offs(pOrigin,375.14,31.32,0.00),v60,z0,tPen\WObj:=wPaper;
    MoveL Offs(pOrigin,370.48,35.98,0.00),v40,fine,tPen\WObj:=wPaper;
    MoveL Offs(pOrigin,370.48,35.98,6.00),v60,z5,tPen\WObj:=wPaper;
    MoveL Offs(pOrigin,368.08,35.39,6.00),vTravel,z5,tPen\WObj:=wPaper;
    MoveL Offs(pOrigin,368.08,35.39,0.00),v60,z0,tPen\WObj:=wPaper;
    MoveL Offs(pOrigin,372.59,30.88,0.00),v40,z0,tPen\WObj:=wPaper;
    MoveL Offs(pOrigin,372.61,31.90,0.00),v40,z0,tPen\WObj:=wPaper;
    MoveL Offs(pOrigin,361.99,31.90,0.00),v40,z0,tPen\WObj:=wPaper;
    MoveL Offs(pOrigin,361.80,32.71,0.00),v40,z0,tPen\WObj:=wPaper;
    MoveL Offs(pOrigin,364.65,29.85,0.00),v40,z0,tPen\WObj:=wPaper;
    MoveL Offs(pOrigin,364.75,30.84,0.00),v40,z0,tPen\WObj:=wPaper;
    MoveL Offs(pOrigin,359.65,30.84,0.00),v40,z0,tPen\WObj:=wPaper;
    MoveL Offs(pOrigin,359.71,31.82,0.00),v40,z0,tPen\WObj:=wPaper;
    MoveL Offs(pOrigin,362.26,29.26,0.00),v40,fine,tPen\WObj:=wPaper;
    MoveL Offs(pOrigin,362.26,29.26,6.00),v60,z5,tPen\WObj:=wPaper;
    MoveL Offs(pOrigin,361.06,28.97,6.00),vTravel,z5,tPen\WObj:=wPaper;
    MoveL Offs(pOrigin,361.06,28.97,0.00),v60,z0,tPen\WObj:=wPaper;
    MoveL Offs(pOrigin,358.51,31.52,0.00),v40,fine,tPen\WObj:=wPaper;
    MoveL Offs(pOrigin,358.51,31.52,6.00),v60,z5,tPen\WObj:=wPaper;
    MoveL Offs(pOrigin,363.28,31.14,6.00),vTravel,z5,tPen\WObj:=wPaper;
    MoveL Offs(pOrigin,363.28,31.14,0.00),v60,z0,tPen\WObj:=wPaper;
    MoveL Offs(pOrigin,363.28,32.20,0.00),v40,z0,tPen\WObj:=wPaper;
    MoveL Offs(pOrigin,364.33,32.62,0.00),v40,z0,tPen\WObj:=wPaper;
    MoveL Offs(pOrigin,364.33,31.35,0.00),v40,z0,tPen\WObj:=wPaper;
    MoveL Offs(pOrigin,365.39,31.56,0.00),v40,z0,tPen\WObj:=wPaper;
    MoveL Offs(pOrigin,365.39,32.84,0.00),v40,fine,tPen\WObj:=wPaper;
    MoveL Offs(pOrigin,365.39,32.84,6.00),v60,z5,tPen\WObj:=wPaper;
    MoveL Offs(pOrigin,354.30,35.73,6.00),vTravel,z5,tPen\WObj:=wPaper;
    MoveL Offs(pOrigin,354.30,35.73,0.00),v60,z0,tPen\WObj:=wPaper;
    MoveL Offs(pOrigin,353.40,36.63,0.00),v40,z0,tPen\WObj:=wPaper;
    MoveL Offs(pOrigin,352.95,35.58,0.00),v40,z0,tPen\WObj:=wPaper;
    MoveL Offs(pOrigin,353.85,34.68,0.00),v40,fine,tPen\WObj:=wPaper;
    MoveL Offs(pOrigin,353.85,34.68,6.00),v60,z5,tPen\WObj:=wPaper;
    MoveL Offs(pOrigin,354.60,36.93,6.00),vTravel,z5,tPen\WObj:=wPaper;
    MoveL Offs(pOrigin,354.60,36.93,0.00),v60,z0,tPen\WObj:=wPaper;
    MoveL Offs(pOrigin,353.69,37.83,0.00),v40,fine,tPen\WObj:=wPaper;
    MoveL Offs(pOrigin,353.69,37.83,6.00),v60,z5,tPen\WObj:=wPaper;
    MoveL Offs(pOrigin,349.82,29.75,6.00),vTravel,z5,tPen\WObj:=wPaper;
    MoveL Offs(pOrigin,349.82,29.75,0.00),v60,z0,tPen\WObj:=wPaper;
    MoveL Offs(pOrigin,345.02,34.56,0.00),v40,fine,tPen\WObj:=wPaper;
    MoveL Offs(pOrigin,345.02,34.56,6.00),v60,z5,tPen\WObj:=wPaper;
    MoveL Offs(pOrigin,347.75,30.29,6.00),vTravel,z5,tPen\WObj:=wPaper;
    MoveL Offs(pOrigin,347.75,30.29,0.00),v60,z0,tPen\WObj:=wPaper;
    MoveL Offs(pOrigin,347.96,30.71,0.00),v40,z0,tPen\WObj:=wPaper;
    MoveL Offs(pOrigin,347.75,30.29,0.00),v40,fine,tPen\WObj:=wPaper;
    MoveL Offs(pOrigin,347.75,30.29,6.00),v60,z5,tPen\WObj:=wPaper;
    MoveL Offs(pOrigin,348.60,29.23,6.00),vTravel,z5,tPen\WObj:=wPaper;
    MoveL Offs(pOrigin,348.60,29.23,0.00),v60,z0,tPen\WObj:=wPaper;
    MoveL Offs(pOrigin,348.81,29.65,0.00),v40,z0,tPen\WObj:=wPaper;
    MoveL Offs(pOrigin,348.60,29.23,0.00),v40,fine,tPen\WObj:=wPaper;
    MoveL Offs(pOrigin,348.60,29.23,6.00),v60,z5,tPen\WObj:=wPaper;
    MoveL Offs(pOrigin,346.05,28.16,6.00),vTravel,z5,tPen\WObj:=wPaper;
    MoveL Offs(pOrigin,346.05,28.16,0.00),v60,z0,tPen\WObj:=wPaper;
    MoveL Offs(pOrigin,346.48,28.59,0.00),v40,z0,tPen\WObj:=wPaper;
    MoveL Offs(pOrigin,346.05,28.16,0.00),v40,fine,tPen\WObj:=wPaper;
    MoveL Offs(pOrigin,346.05,28.16,6.00),v60,z5,tPen\WObj:=wPaper;
    MoveL Offs(pOrigin,346.05,26.67,6.00),vTravel,z5,tPen\WObj:=wPaper;
    MoveL Offs(pOrigin,346.05,26.67,0.00),v60,z0,tPen\WObj:=wPaper;
    MoveL Offs(pOrigin,347.54,27.95,0.00),v40,z0,tPen\WObj:=wPaper;
    MoveL Offs(pOrigin,346.05,26.67,0.00),v40,fine,tPen\WObj:=wPaper;
    MoveL Offs(pOrigin,346.05,26.67,6.00),v60,z5,tPen\WObj:=wPaper;
    MoveL Offs(pOrigin,347.43,26.64,6.00),vTravel,z5,tPen\WObj:=wPaper;
    MoveL Offs(pOrigin,347.43,26.64,0.00),v60,z0,tPen\WObj:=wPaper;
    MoveL Offs(pOrigin,344.57,23.78,0.00),v40,z0,tPen\WObj:=wPaper;
    MoveL Offs(pOrigin,344.45,23.18,0.00),v40,z0,tPen\WObj:=wPaper;
    MoveL Offs(pOrigin,337.54,30.09,0.00),v40,z0,tPen\WObj:=wPaper;
    MoveL Offs(pOrigin,338.59,30.53,0.00),v40,z0,tPen\WObj:=wPaper;
    MoveL Offs(pOrigin,345.80,23.32,0.00),v40,fine,tPen\WObj:=wPaper;
    MoveL Offs(pOrigin,345.80,23.32,6.00),v60,z5,tPen\WObj:=wPaper;
    MoveL Offs(pOrigin,347.00,23.62,6.00),vTravel,z5,tPen\WObj:=wPaper;
    MoveL Offs(pOrigin,347.00,23.62,0.00),v60,z0,tPen\WObj:=wPaper;
    MoveL Offs(pOrigin,339.78,30.83,0.00),v40,z0,tPen\WObj:=wPaper;
    MoveL Offs(pOrigin,339.05,30.21,0.00),v40,z0,tPen\WObj:=wPaper;
    MoveL Offs(pOrigin,334.69,25.85,0.00),v40,z0,tPen\WObj:=wPaper;
    MoveL Offs(pOrigin,334.77,26.89,0.00),v40,z0,tPen\WObj:=wPaper;
    MoveL Offs(pOrigin,334.77,28.16,0.00),v40,fine,tPen\WObj:=wPaper;
    MoveL Offs(pOrigin,334.77,28.16,6.00),v60,z5,tPen\WObj:=wPaper;
    MoveL Offs(pOrigin,332.45,29.20,6.00),vTravel,z5,tPen\WObj:=wPaper;
    MoveL Offs(pOrigin,332.45,29.20,0.00),v60,z0,tPen\WObj:=wPaper;
  ENDPROC

